LIN {X 0,Y 523.94,Z 179.22,A -85,B 0,C 180,E1 -4815.311,E2 -4815.311} C_VEL
LIN {X 0,Y 523.942,Z 179.221,A -85,B 0,C 180,E1 -4818.692,E2 -4818.692} C_VEL
LIN {X 0,Y 523.916,Z 179.219,A -85,B 0,C 180,E1 -4821.898,E2 -4821.898} C_VEL
LIN {X 0,Y 523.925,Z 179.226,A -85,B 0,C 180,E1 -4824.911,E2 -4824.911} C_VEL
LIN {X 0,Y 523.936,Z 179.217,A -85,B 0,C 180,E1 -4827.68,E2 -4827.68} C_VEL
LIN {X 0,Y 523.955,Z 179.221,A -85,B 0,C 180,E1 -4830.677,E2 -4830.677} C_VEL
LIN {X 0,Y 523.973,Z 179.213,A -85,B 0,C 180,E1 -4833.728,E2 -4833.728} C_VEL
LIN {X 0,Y 523.914,Z 179.223,A -85,B 0,C 180,E1 -4836.269,E2 -4836.269} C_VEL
LIN {X 0,Y 523.947,Z 179.222,A -85,B 0,C 180,E1 -4838.766,E2 -4838.766} C_VEL
LIN {X 0,Y 523.941,Z 179.218,A -85,B 0,C 180,E1 -4841.22,E2 -4841.22} C_VEL
LIN {X 0,Y 523.928,Z 179.219,A -85,B 0,C 180,E1 -4843.638,E2 -4843.638} C_VEL
LIN {X 0,Y 523.935,Z 179.221,A -85,B 0,C 180,E1 -4846.028,E2 -4846.028} C_VEL
LIN {X 0,Y 523.995,Z 179.211,A -85,B 0,C 180,E1 -4849.177,E2 -4849.177} C_VEL
LIN {X 0,Y 524.008,Z 179.216,A -85,B 0,C 180,E1 -4852.292,E2 -4852.292} C_VEL
LIN {X 0,Y 524.075,Z 179.206,A -85,B 0,C 180,E1 -4854.613,E2 -4854.613} C_VEL
LIN {X 0,Y 524.109,Z 179.2,A -85,B 0,C 180,E1 -4857.694,E2 -4857.694} C_VEL
LIN {X 0,Y 524.051,Z 179.302,A -85,B 0,C 180,E1 -4860.264,E2 -4860.264} C_VEL
LIN {X 0,Y 524.006,Z 197.303,A -85,B 0,C 180,E1 -4863.267,E2 -4863.267} C_VEL
LIN {X 0,Y 524.025,Z 211.019,A -85,B 0,C 180,E1 -4865.58,E2 -4865.58} C_VEL
LIN {X 0,Y 524.022,Z 224.908,A -85,B 0,C 180,E1 -4867.995,E2 -4867.995} C_VEL
LIN {X 0,Y 525.186,Z 232.663,A -85,B 0,C 180,E1 -4868.169,E2 -4868.169} C_VEL
LIN {X 0,Y 524.869,Z 303.638,A -85,B 0,C 180,E1 -4869.222,E2 -4869.222} C_VEL
LIN {X 0,Y 524.725,Z 315.282,A -85,B 0,C 180,E1 -4869.54,E2 -4869.54} C_VEL
LIN {X 0,Y 524.579,Z 326.858,A -85,B 0,C 180,E1 -4870.03,E2 -4870.03} C_VEL
LIN {X 0,Y 524.417,Z 337.03,A -85,B 0,C 180,E1 -4870.618,E2 -4870.618} C_VEL
LIN {X 0,Y 524.207,Z 347.39,A -85,B 0,C 180,E1 -4871.405,E2 -4871.405} C_VEL
LIN {X 0,Y 524.042,Z 355.429,A -85,B 0,C 180,E1 -4872.186,E2 -4872.186} C_VEL
LIN {X 0,Y 523.848,Z 363.637,A -85,B 0,C 180,E1 -4873.183,E2 -4873.183} C_VEL
LIN {X 0,Y 523.764,Z 370.012,A -85,B 0,C 180,E1 -4874.175,E2 -4874.175} C_VEL
LIN {X 0,Y 523.63,Z 375.152,A -85,B 0,C 180,E1 -4875.183,E2 -4875.183} C_VEL
LIN {X 0,Y 523.55,Z 379.695,A -85,B 0,C 180,E1 -4876.373,E2 -4876.373} C_VEL
LIN {X 0,Y 523.437,Z 382.89,A -85,B 0,C 180,E1 -4877.581,E2 -4877.581} C_VEL
LIN {X 0,Y 523.414,Z 384.762,A -85,B 0,C 180,E1 -4878.799,E2 -4878.799} C_VEL
LIN {X 0,Y 523.414,Z 385.391,A -85,B 0,C 180,E1 -4879.964,E2 -4879.964} C_VEL
LIN {X 0,Y 523.385,Z 384.744,A -85,B 0,C 180,E1 -4881.257,E2 -4881.257} C_VEL
LIN {X 0,Y 523.433,Z 383.554,A -85,B 0,C 180,E1 -4882.113,E2 -4882.113} C_VEL
LIN {X 0,Y 523.469,Z 380.727,A -85,B 0,C 180,E1 -4883.332,E2 -4883.332} C_VEL
LIN {X 0,Y 523.595,Z 376.321,A -85,B 0,C 180,E1 -4884.588,E2 -4884.588} C_VEL
LIN {X 0,Y 523.693,Z 371.04,A -85,B 0,C 180,E1 -4885.693,E2 -4885.693} C_VEL
LIN {X 0,Y 523.788,Z 364.719,A -85,B 0,C 180,E1 -4886.711,E2 -4886.711} C_VEL
LIN {X 0,Y 523.948,Z 356.846,A -85,B 0,C 180,E1 -4887.712,E2 -4887.712} C_VEL
LIN {X 0,Y 524.148,Z 347.477,A -85,B 0,C 180,E1 -4888.643,E2 -4888.643} C_VEL
LIN {X 0,Y 524.349,Z 337.621,A -85,B 0,C 180,E1 -4889.4,E2 -4889.4} C_VEL
LIN {X 0,Y 524.512,Z 327.606,A -85,B 0,C 180,E1 -4889.996,E2 -4889.996} C_VEL
LIN {X 0,Y 524.704,Z 315.795,A -85,B 0,C 180,E1 -4890.507,E2 -4890.507} C_VEL
LIN {X 0,Y 524.112,Z 310.181,A -85,B 0,C 180,E1 -4890.703,E2 -4890.703} C_VEL
LIN {X 0,Y 521.241,Z 300.997,A -85,B 0,C 180,E1 -4890.982,E2 -4890.982} C_VEL
LIN {X 0,Y 518.404,Z 291.68,A -85,B 0,C 180,E1 -4891.192,E2 -4891.192} C_VEL
LIN {X 0,Y 517.926,Z 285.863,A -85,B 0,C 180,E1 -4891.284,E2 -4891.284} C_VEL
LIN {X 0,Y 518.086,Z 231.937,A -85,B 0,C 180,E1 -4892.071,E2 -4892.071} C_VEL
LIN {X 0,Y 516.963,Z 225.027,A -85,B 0,C 180,E1 -4892.227,E2 -4892.227} C_VEL
LIN {X 0,Y 516.978,Z 220.993,A -85,B 0,C 180,E1 -4892.941,E2 -4892.941} C_VEL
LIN {X 0,Y 517.185,Z 204.967,A -85,B 0,C 180,E1 -4895.995,E2 -4895.995} C_VEL
LIN {X 0,Y 517.364,Z 187.914,A -85,B 0,C 180,E1 -4899.258,E2 -4899.258} C_VEL
LIN {X 0,Y 517.251,Z 181.728,A -85,B 0,C 180,E1 -4900.458,E2 -4900.458} C_VEL
LIN {X 0,Y 516.952,Z 180.119,A -85,B 0,C 180,E1 -4900.847,E2 -4900.847} C_VEL
LIN {X 0,Y 516.88,Z 180.104,A -85,B 0,C 180,E1 -4903.903,E2 -4903.903} C_VEL
LIN {X 0,Y 516.88,Z 180.101,A -85,B 0,C 180,E1 -4906.107,E2 -4906.107} C_VEL
LIN {X 0,Y 516.913,Z 180.092,A -85,B 0,C 180,E1 -4908.398,E2 -4908.398} C_VEL
LIN {X 0,Y 516.879,Z 180.099,A -85,B 0,C 180,E1 -4911.284,E2 -4911.284} C_VEL
LIN {X 0,Y 516.886,Z 180.096,A -85,B 0,C 180,E1 -4914.221,E2 -4914.221} C_VEL
LIN {X 0,Y 516.893,Z 180.095,A -85,B 0,C 180,E1 -4917.053,E2 -4917.053} C_VEL
LIN {X 0,Y 516.89,Z 180.099,A -85,B 0,C 180,E1 -4919.796,E2 -4919.796} C_VEL
LIN {X 0,Y 516.928,Z 180.089,A -85,B 0,C 180,E1 -4922.467,E2 -4922.467} C_VEL
LIN {X 0,Y 516.909,Z 180.095,A -85,B 0,C 180,E1 -4925.071,E2 -4925.071} C_VEL
LIN {X 0,Y 516.884,Z 180.094,A -85,B 0,C 180,E1 -4928.462,E2 -4928.462} C_VEL
LIN {X 0,Y 516.9,Z 180.096,A -85,B 0,C 180,E1 -4930.954,E2 -4930.954} C_VEL
LIN {X 0,Y 516.913,Z 180.099,A -85,B 0,C 180,E1 -4933.41,E2 -4933.41} C_VEL
LIN {X 0,Y 516.904,Z 180.094,A -85,B 0,C 180,E1 -4935.833,E2 -4935.833} C_VEL
LIN {X 0,Y 516.95,Z 180.092,A -85,B 0,C 180,E1 -4939.027,E2 -4939.027} C_VEL
LIN {X 0,Y 516.977,Z 180.083,A -85,B 0,C 180,E1 -4942.186,E2 -4942.186} C_VEL
LIN {X 0,Y 517.032,Z 180.077,A -85,B 0,C 180,E1 -4944.54,E2 -4944.54} C_VEL
LIN {X 0,Y 517.083,Z 180.072,A -85,B 0,C 180,E1 -4947.663,E2 -4947.663} C_VEL
LIN {X 0,Y 517.091,Z 180.073,A -85,B 0,C 180,E1 -4950.778,E2 -4950.778} C_VEL
LIN {X 0,Y 517.011,Z 180.087,A -85,B 0,C 180,E1 -4953.116,E2 -4953.116} C_VEL
LIN {X 0,Y 517,Z 180.081,A -85,B 0,C 180,E1 -4956.243,E2 -4956.243} C_VEL
LIN {X 0,Y 516.95,Z 180.089,A -85,B 0,C 180,E1 -4959.389,E2 -4959.389} C_VEL
LIN {X 0,Y 516.949,Z 180.086,A -85,B 0,C 180,E1 -4961.807,E2 -4961.807} C_VEL
LIN {X 0,Y 516.94,Z 180.092,A -85,B 0,C 180,E1 -4965.146,E2 -4965.146} C_VEL
LIN {X 0,Y 516.921,Z 180.092,A -85,B 0,C 180,E1 -4968.222,E2 -4968.222} C_VEL
LIN {X 0,Y 516.908,Z 180.1,A -85,B 0,C 180,E1 -4970.701,E2 -4970.701} C_VEL
LIN {X 0,Y 516.906,Z 180.093,A -85,B 0,C 180,E1 -4974.071,E2 -4974.071} C_VEL
LIN {X 0,Y 516.924,Z 180.099,A -85,B 0,C 180,E1 -4976.657,E2 -4976.657} C_VEL
LIN {X 0,Y 516.906,Z 180.092,A -85,B 0,C 180,E1 -4979.523,E2 -4979.523} C_VEL
LIN {X 0,Y 516.895,Z 180.102,A -85,B 0,C 180,E1 -4982.544,E2 -4982.544} C_VEL
LIN {X 0,Y 516.877,Z 180.096,A -85,B 0,C 180,E1 -4985.332,E2 -4985.332} C_VEL
LIN {X 0,Y 516.875,Z 180.098,A -85,B 0,C 180,E1 -4987.943,E2 -4987.943} C_VEL
LIN {X 0,Y 516.897,Z 180.098,A -85,B 0,C 180,E1 -4990.739,E2 -4990.739} C_VEL
LIN {X 0,Y 516.875,Z 180.098,A -85,B 0,C 180,E1 -4993.903,E2 -4993.903} C_VEL
LIN {X 0,Y 516.874,Z 180.101,A -85,B 0,C 180,E1 -4996.107,E2 -4996.107} C_VEL
LIN {X 0,Y 516.896,Z 180.093,A -85,B 0,C 180,E1 -4999.26,E2 -4999.26} C_VEL
LIN {X 0,Y 516.857,Z 180.107,A -85,B 0,C 180,E1 -5002.274,E2 -5002.274} C_VEL
LIN {X 0,Y 516.888,Z 180.094,A -85,B 0,C 180,E1 -5005.176,E2 -5005.176} C_VEL
LIN {X 0,Y 516.876,Z 180.102,A -85,B 0,C 180,E1 -5007.976,E2 -5007.976} C_VEL
LIN {X 0,Y 516.928,Z 180.091,A -85,B 0,C 180,E1 -5010.696,E2 -5010.696} C_VEL
LIN {X 0,Y 516.934,Z 180.093,A -85,B 0,C 180,E1 -5013.804,E2 -5013.804} C_VEL
LIN {X 0,Y 516.863,Z 180.098,A -85,B 0,C 180,E1 -5016.777,E2 -5016.777} C_VEL
LIN {X 0,Y 516.931,Z 180.094,A -85,B 0,C 180,E1 -5019.731,E2 -5019.731} C_VEL
LIN {X 0,Y 516.922,Z 180.091,A -85,B 0,C 180,E1 -5022.596,E2 -5022.596} C_VEL
LIN {X 0,Y 516.933,Z 180.089,A -85,B 0,C 180,E1 -5025.03,E2 -5025.03} C_VEL
LIN {X 0,Y 516.956,Z 180.089,A -85,B 0,C 180,E1 -5028.234,E2 -5028.234} C_VEL
LIN {X 0,Y 516.961,Z 180.088,A -85,B 0,C 180,E1 -5031.4,E2 -5031.4} C_VEL
LIN {X 0,Y 517,Z 180.089,A -85,B 0,C 180,E1 -5033.757,E2 -5033.757} C_VEL
LIN {X 0,Y 517.074,Z 180.079,A -85,B 0,C 180,E1 -5037.663,E2 -5037.663} C_VEL
LIN {X 0,Y 517.085,Z 180.069,A -85,B 0,C 180,E1 -5040.779,E2 -5040.779} C_VEL
LIN {X 0,Y 517.006,Z 180.082,A -85,B 0,C 180,E1 -5043.117,E2 -5043.117} C_VEL
LIN {X 0,Y 516.994,Z 180.082,A -85,B 0,C 180,E1 -5046.244,E2 -5046.244} C_VEL
LIN {X 0,Y 516.941,Z 180.094,A -85,B 0,C 180,E1 -5049.39,E2 -5049.39} C_VEL
LIN {X 0,Y 516.944,Z 180.091,A -85,B 0,C 180,E1 -5051.807,E2 -5051.807} C_VEL
LIN {X 0,Y 516.937,Z 180.093,A -85,B 0,C 180,E1 -5055.147,E2 -5055.147} C_VEL
LIN {X 0,Y 516.917,Z 180.091,A -85,B 0,C 180,E1 -5058.223,E2 -5058.223} C_VEL
LIN {X 0,Y 516.905,Z 180.093,A -85,B 0,C 180,E1 -5060.702,E2 -5060.702} C_VEL
LIN {X 0,Y 516.884,Z 180.095,A -85,B 0,C 180,E1 -5064.074,E2 -5064.074} C_VEL
LIN {X 0,Y 516.917,Z 180.092,A -85,B 0,C 180,E1 -5066.659,E2 -5066.659} C_VEL
LIN {X 0,Y 516.903,Z 180.097,A -85,B 0,C 180,E1 -5069.524,E2 -5069.524} C_VEL
LIN {X 0,Y 516.888,Z 180.095,A -85,B 0,C 180,E1 -5072.544,E2 -5072.544} C_VEL
LIN {X 0,Y 516.86,Z 180.103,A -85,B 0,C 180,E1 -5075.33,E2 -5075.33} C_VEL
LIN {X 0,Y 516.874,Z 180.096,A -85,B 0,C 180,E1 -5077.944,E2 -5077.944} C_VEL
LIN {X 0,Y 516.878,Z 180.1,A -85,B 0,C 180,E1 -5080.743,E2 -5080.743} C_VEL
LIN {X 0,Y 516.878,Z 180.102,A -85,B 0,C 180,E1 -5082.832,E2 -5082.832} C_VEL
LIN {X 0,Y 516.919,Z 180.099,A -85,B 0,C 180,E1 -5085.011,E2 -5085.011} C_VEL
LIN {X 0,Y 516.899,Z 180.095,A -85,B 0,C 180,E1 -5088.401,E2 -5088.401} C_VEL
LIN {X 0,Y 516.877,Z 180.099,A -85,B 0,C 180,E1 -5091.285,E2 -5091.285} C_VEL
LIN {X 0,Y 516.865,Z 180.098,A -85,B 0,C 180,E1 -5094.22,E2 -5094.22} C_VEL
LIN {X 0,Y 516.893,Z 180.101,A -85,B 0,C 180,E1 -5097.054,E2 -5097.054} C_VEL
LIN {X 0,Y 516.881,Z 180.098,A -85,B 0,C 180,E1 -5099.797,E2 -5099.797} C_VEL
LIN {X 0,Y 516.898,Z 180.101,A -85,B 0,C 180,E1 -5102.467,E2 -5102.467} C_VEL
LIN {X 0,Y 516.915,Z 180.238,A -85,B 0,C 180,E1 -5104.05,E2 -5104.05} C_VEL
LIN {X 0,Y 519.406,Z 191.693,A -85,B 0,C 180,E1 -5105.627,E2 -5105.627} C_VEL
LIN {X 0,Y 518.761,Z 215.518,A -85,B 0,C 180,E1 -5108.545,E2 -5108.545} C_VEL
LIN {X 0,Y 518.012,Z 242.728,A -85,B 0,C 180,E1 -5111.818,E2 -5111.818} C_VEL
LIN {X 0,Y 517.52,Z 267.094,A -85,B 0,C 180,E1 -5114.703,E2 -5114.703} C_VEL
LIN {X 0,Y 518.203,Z 273.127,A -85,B 0,C 180,E1 -5114.84,E2 -5114.84} C_VEL
LIN {X 0,Y 518.795,Z 280.471,A -85,B 0,C 180,E1 -5114.962,E2 -5114.962} C_VEL
LIN {X 0,Y 518.343,Z 376.522,A -85,B 0,C 180,E1 -5116.325,E2 -5116.325} C_VEL
LIN {X 0,Y 518.146,Z 389.838,A -85,B 0,C 180,E1 -5116.669,E2 -5116.669} C_VEL
LIN {X 0,Y 517.889,Z 402.606,A -85,B 0,C 180,E1 -5117.161,E2 -5117.161} C_VEL
LIN {X 0,Y 517.597,Z 414.328,A -85,B 0,C 180,E1 -5117.777,E2 -5117.777} C_VEL
LIN {X 0,Y 517.332,Z 425.652,A -85,B 0,C 180,E1 -5118.541,E2 -5118.541} C_VEL
LIN {X 0,Y 517.043,Z 436.193,A -85,B 0,C 180,E1 -5119.427,E2 -5119.427} C_VEL
LIN {X 0,Y 516.816,Z 445.668,A -85,B 0,C 180,E1 -5120.411,E2 -5120.411} C_VEL
LIN {X 0,Y 516.626,Z 454.821,A -85,B 0,C 180,E1 -5121.592,E2 -5121.592} C_VEL
LIN {X 0,Y 516.502,Z 462.192,A -85,B 0,C 180,E1 -5122.77,E2 -5122.77} C_VEL
LIN {X 0,Y 516.383,Z 467.166,A -85,B 0,C 180,E1 -5123.75,E2 -5123.75} C_VEL
LIN {X 0,Y 516.312,Z 471.994,A -85,B 0,C 180,E1 -5124.925,E2 -5124.925} C_VEL
LIN {X 0,Y 516.372,Z 475.691,A -85,B 0,C 180,E1 -5126.099,E2 -5126.099} C_VEL
LIN {X 0,Y 516.382,Z 477.594,A -85,B 0,C 180,E1 -5126.88,E2 -5126.88} C_VEL
LIN {X 0,Y 516.272,Z 479.011,A -85,B 0,C 180,E1 -5127.66,E2 -5127.66} C_VEL
LIN {X 0,Y 516.23,Z 480.634,A -85,B 0,C 180,E1 -5129.221,E2 -5129.221} C_VEL
LIN {X 0,Y 516.235,Z 480.847,A -85,B 0,C 180,E1 -5130.001,E2 -5130.001} C_VEL
LIN {X 0,Y 516.231,Z 480.617,A -85,B 0,C 180,E1 -5130.781,E2 -5130.781} C_VEL
LIN {X 0,Y 516.235,Z 479.989,A -85,B 0,C 180,E1 -5131.561,E2 -5131.561} C_VEL
LIN {X 0,Y 516.275,Z 478.962,A -85,B 0,C 180,E1 -5132.341,E2 -5132.341} C_VEL
LIN {X 0,Y 516.383,Z 477.526,A -85,B 0,C 180,E1 -5133.121,E2 -5133.121} C_VEL
LIN {X 0,Y 516.365,Z 474.5,A -85,B 0,C 180,E1 -5134.294,E2 -5134.294} C_VEL
LIN {X 0,Y 516.4,Z 470.409,A -85,B 0,C 180,E1 -5135.467,E2 -5135.467} C_VEL
LIN {X 0,Y 516.442,Z 465.064,A -85,B 0,C 180,E1 -5136.656,E2 -5136.656} C_VEL
LIN {X 0,Y 516.544,Z 458.49,A -85,B 0,C 180,E1 -5137.82,E2 -5137.82} C_VEL
LIN {X 0,Y 516.707,Z 450.22,A -85,B 0,C 180,E1 -5138.999,E2 -5138.999} C_VEL
LIN {X 0,Y 516.865,Z 441.765,A -85,B 0,C 180,E1 -5139.984,E2 -5139.984} C_VEL
LIN {X 0,Y 517.179,Z 431.397,A -85,B 0,C 180,E1 -5140.968,E2 -5140.968} C_VEL
LIN {X 0,Y 517.443,Z 419.886,A -85,B 0,C 180,E1 -5141.839,E2 -5141.839} C_VEL
LIN {X 0,Y 517.699,Z 408.046,A -85,B 0,C 180,E1 -5142.545,E2 -5142.545} C_VEL
LIN {X 0,Y 518.002,Z 396.026,A -85,B 0,C 180,E1 -5143.086,E2 -5143.086} C_VEL
LIN {X 0,Y 518.211,Z 383,A -85,B 0,C 180,E1 -5143.505,E2 -5143.505} C_VEL
LIN {X 0,Y 518.386,Z 370.827,A -85,B 0,C 180,E1 -5143.75,E2 -5143.75} C_VEL
LIN {X 0,Y 518.619,Z 277.097,A -85,B 0,C 180,E1 -5145.075,E2 -5145.075} C_VEL
LIN {X 0,Y 517.474,Z 266.884,A -85,B 0,C 180,E1 -5145.268,E2 -5145.268} C_VEL
LIN {X 0,Y 517.95,Z 241.231,A -85,B 0,C 180,E1 -5148.227,E2 -5148.227} C_VEL
LIN {X 0,Y 518.556,Z 211.729,A -85,B 0,C 180,E1 -5151.674,E2 -5151.674} C_VEL
LIN {X 0,Y 518.97,Z 190.784,A -85,B 0,C 180,E1 -5154.152,E2 -5154.152} C_VEL
LIN {X 0,Y 516.921,Z 180.235,A -85,B 0,C 180,E1 -5155.533,E2 -5155.533} C_VEL
LIN {X 0,Y 516.855,Z 180.103,A -85,B 0,C 180,E1 -5158.419,E2 -5158.419} C_VEL
LIN {X 0,Y 516.89,Z 180.103,A -85,B 0,C 180,E1 -5161.11,E2 -5161.11} C_VEL
LIN {X 0,Y 516.888,Z 180.097,A -85,B 0,C 180,E1 -5163.962,E2 -5163.962} C_VEL
LIN {X 0,Y 516.856,Z 180.104,A -85,B 0,C 180,E1 -5166.748,E2 -5166.748} C_VEL
LIN {X 0,Y 516.861,Z 180.101,A -85,B 0,C 180,E1 -5169.724,E2 -5169.724} C_VEL
LIN {X 0,Y 516.887,Z 180.097,A -85,B 0,C 180,E1 -5171.778,E2 -5171.778} C_VEL
LIN {X 0,Y 516.898,Z 180.102,A -85,B 0,C 180,E1 -5175.007,E2 -5175.007} C_VEL
LIN {X 0,Y 516.905,Z 180.094,A -85,B 0,C 180,E1 -5178.4,E2 -5178.4} C_VEL
LIN {X 0,Y 516.881,Z 180.099,A -85,B 0,C 180,E1 -5181.284,E2 -5181.284} C_VEL
LIN {X 0,Y 516.873,Z 180.098,A -85,B 0,C 180,E1 -5184.219,E2 -5184.219} C_VEL
LIN {X 0,Y 516.883,Z 180.101,A -85,B 0,C 180,E1 -5187.052,E2 -5187.052} C_VEL
LIN {X 0,Y 516.888,Z 180.095,A -85,B 0,C 180,E1 -5189.796,E2 -5189.796} C_VEL
LIN {X 0,Y 516.924,Z 180.097,A -85,B 0,C 180,E1 -5192.467,E2 -5192.467} C_VEL
LIN {X 0,Y 516.874,Z 180.1,A -85,B 0,C 180,E1 -5195.07,E2 -5195.07} C_VEL
LIN {X 0,Y 516.871,Z 180.097,A -85,B 0,C 180,E1 -5197.621,E2 -5197.621} C_VEL
LIN {X 0,Y 516.931,Z 180.093,A -85,B 0,C 180,E1 -5200.129,E2 -5200.129} C_VEL
LIN {X 0,Y 516.898,Z 180.101,A -85,B 0,C 180,E1 -5202.595,E2 -5202.595} C_VEL
LIN {X 0,Y 516.944,Z 180.091,A -85,B 0,C 180,E1 -5205.03,E2 -5205.03} C_VEL
LIN {X 0,Y 516.967,Z 180.091,A -85,B 0,C 180,E1 -5208.233,E2 -5208.233} C_VEL
LIN {X 0,Y 516.958,Z 180.087,A -85,B 0,C 180,E1 -5211.399,E2 -5211.399} C_VEL
LIN {X 0,Y 517.022,Z 180.085,A -85,B 0,C 180,E1 -5214.54,E2 -5214.54} C_VEL
LIN {X 0,Y 517.082,Z 180.075,A -85,B 0,C 180,E1 -5217.663,E2 -5217.663} C_VEL
LIN {X 0,Y 517.052,Z 180.202,A -85,B 0,C 180,E1 -5220.194,E2 -5220.194} C_VEL
LIN {X 0,Y 517.03,Z 199.023,A -85,B 0,C 180,E1 -5223.311,E2 -5223.311} C_VEL
LIN {X 0,Y 517.045,Z 214.996,A -85,B 0,C 180,E1 -5226.047,E2 -5226.047} C_VEL
LIN {X 0,Y 517.037,Z 224.992,A -85,B 0,C 180,E1 -5227.785,E2 -5227.785} C_VEL
LIN {X 0,Y 517.424,Z 227.519,A -85,B 0,C 180,E1 -5227.88,E2 -5227.88} C_VEL
LIN {X 0,Y 518.316,Z 234.268,A -85,B 0,C 180,E1 -5228.008,E2 -5228.008} C_VEL
LIN {X 0,Y 517.914,Z 304.483,A -85,B 0,C 180,E1 -5229.076,E2 -5229.076} C_VEL
LIN {X 0,Y 517.771,Z 316.676,A -85,B 0,C 180,E1 -5229.423,E2 -5229.423} C_VEL
LIN {X 0,Y 517.622,Z 328.964,A -85,B 0,C 180,E1 -5229.968,E2 -5229.968} C_VEL
LIN {X 0,Y 517.4,Z 340.176,A -85,B 0,C 180,E1 -5230.665,E2 -5230.665} C_VEL
LIN {X 0,Y 517.208,Z 349.918,A -85,B 0,C 180,E1 -5231.462,E2 -5231.462} C_VEL
LIN {X 0,Y 516.998,Z 358.584,A -85,B 0,C 180,E1 -5232.362,E2 -5232.362} C_VEL
LIN {X 0,Y 516.813,Z 366.175,A -85,B 0,C 180,E1 -5233.366,E2 -5233.366} C_VEL
LIN {X 0,Y 516.681,Z 372.203,A -85,B 0,C 180,E1 -5234.373,E2 -5234.373} C_VEL
LIN {X 0,Y 516.569,Z 376.772,A -85,B 0,C 180,E1 -5235.344,E2 -5235.344} C_VEL
LIN {X 0,Y 516.461,Z 381.227,A -85,B 0,C 180,E1 -5236.604,E2 -5236.604} C_VEL
LIN {X 0,Y 516.388,Z 383.835,A -85,B 0,C 180,E1 -5237.694,E2 -5237.694} C_VEL
LIN {X 0,Y 516.344,Z 385.689,A -85,B 0,C 180,E1 -5239.066,E2 -5239.066} C_VEL
LIN {X 0,Y 516.345,Z 386.049,A -85,B 0,C 180,E1 -5240.089,E2 -5240.089} C_VEL
LIN {X 0,Y 516.32,Z 385.831,A -85,B 0,C 180,E1 -5240.726,E2 -5240.726} C_VEL
LIN {X 0,Y 516.324,Z 385.075,A -85,B 0,C 180,E1 -5241.562,E2 -5241.562} C_VEL
LIN {X 0,Y 516.366,Z 383.7,A -85,B 0,C 180,E1 -5242.401,E2 -5242.401} C_VEL
LIN {X 0,Y 516.45,Z 380.478,A -85,B 0,C 180,E1 -5243.668,E2 -5243.668} C_VEL
LIN {X 0,Y 516.549,Z 375.681,A -85,B 0,C 180,E1 -5244.946,E2 -5244.946} C_VEL
LIN {X 0,Y 516.678,Z 369.555,A -85,B 0,C 180,E1 -5246.136,E2 -5246.136} C_VEL
LIN {X 0,Y 516.826,Z 363.178,A -85,B 0,C 180,E1 -5247.1,E2 -5247.1} C_VEL
LIN {X 0,Y 517.017,Z 354.953,A -85,B 0,C 180,E1 -5248.086,E2 -5248.086} C_VEL
LIN {X 0,Y 517.206,Z 345.75,A -85,B 0,C 180,E1 -5248.952,E2 -5248.952} C_VEL
LIN {X 0,Y 517.461,Z 335.624,A -85,B 0,C 180,E1 -5249.695,E2 -5249.695} C_VEL
LIN {X 0,Y 517.642,Z 324.246,A -85,B 0,C 180,E1 -5250.324,E2 -5250.324} C_VEL
LIN {X 0,Y 517.787,Z 312.012,A -85,B 0,C 180,E1 -5250.794,E2 -5250.794} C_VEL
LIN {X 0,Y 517.861,Z 300.164,A -85,B 0,C 180,E1 -5251.074,E2 -5251.074} C_VEL
LIN {X 0,Y 517.926,Z 285.863,A -85,B 0,C 180,E1 -5251.284,E2 -5251.284} C_VEL
LIN {X 0,Y 517.466,Z 280.046,A -85,B 0,C 180,E1 -5251.379,E2 -5251.379} C_VEL
LIN {X 0,Y 514.659,Z 270.702,A -85,B 0,C 180,E1 -5251.584,E2 -5251.584} C_VEL
LIN {X 0,Y 511.765,Z 261.363,A -85,B 0,C 180,E1 -5251.796,E2 -5251.796} C_VEL
LIN {X 0,Y 511.163,Z 255.544,A -85,B 0,C 180,E1 -5251.899,E2 -5251.899} C_VEL
LIN {X 0,Y 511.211,Z 232.848,A -85,B 0,C 180,E1 -5252.241,E2 -5252.241} C_VEL
LIN {X 0,Y 509.952,Z 225.174,A -85,B 0,C 180,E1 -5252.418,E2 -5252.418} C_VEL
LIN {X 0,Y 510.076,Z 210.803,A -85,B 0,C 180,E1 -5255.116,E2 -5255.116} C_VEL
LIN {X 0,Y 510.248,Z 196.891,A -85,B 0,C 180,E1 -5257.792,E2 -5257.792} C_VEL
LIN {X 0,Y 510.38,Z 183.783,A -85,B 0,C 180,E1 -5260.33,E2 -5260.33} C_VEL
LIN {X 0,Y 509.903,Z 181,A -85,B 0,C 180,E1 -5260.945,E2 -5260.945} C_VEL
LIN {X 0,Y 509.82,Z 180.98,A -85,B 0,C 180,E1 -5264.206,E2 -5264.206} C_VEL
LIN {X 0,Y 509.821,Z 180.976,A -85,B 0,C 180,E1 -5266.937,E2 -5266.937} C_VEL
LIN {X 0,Y 509.837,Z 180.98,A -85,B 0,C 180,E1 -5269.617,E2 -5269.617} C_VEL
LIN {X 0,Y 509.817,Z 180.975,A -85,B 0,C 180,E1 -5272.659,E2 -5272.659} C_VEL
LIN {X 0,Y 509.858,Z 180.976,A -85,B 0,C 180,E1 -5275.796,E2 -5275.796} C_VEL
LIN {X 0,Y 509.844,Z 180.972,A -85,B 0,C 180,E1 -5278.72,E2 -5278.72} C_VEL
LIN {X 0,Y 509.897,Z 180.968,A -85,B 0,C 180,E1 -5281.899,E2 -5281.899} C_VEL
LIN {X 0,Y 509.876,Z 180.968,A -85,B 0,C 180,E1 -5284.704,E2 -5284.704} C_VEL
LIN {X 0,Y 509.825,Z 180.983,A -85,B 0,C 180,E1 -5287.457,E2 -5287.457} C_VEL
LIN {X 0,Y 509.915,Z 180.965,A -85,B 0,C 180,E1 -5289.844,E2 -5289.844} C_VEL
LIN {X 0,Y 509.881,Z 180.973,A -85,B 0,C 180,E1 -5293.174,E2 -5293.174} C_VEL
LIN {X 0,Y 509.872,Z 180.972,A -85,B 0,C 180,E1 -5295.634,E2 -5295.634} C_VEL
LIN {X 0,Y 509.912,Z 180.967,A -85,B 0,C 180,E1 -5298.874,E2 -5298.874} C_VEL
LIN {X 0,Y 509.95,Z 180.958,A -85,B 0,C 180,E1 -5302.078,E2 -5302.078} C_VEL
LIN {X 0,Y 509.983,Z 180.955,A -85,B 0,C 180,E1 -5304.464,E2 -5304.464} C_VEL
LIN {X 0,Y 510.054,Z 180.947,A -85,B 0,C 180,E1 -5307.63,E2 -5307.63} C_VEL
LIN {X 0,Y 510.061,Z 180.949,A -85,B 0,C 180,E1 -5310.789,E2 -5310.789} C_VEL
LIN {X 0,Y 509.953,Z 180.965,A -85,B 0,C 180,E1 -5313.16,E2 -5313.16} C_VEL
LIN {X 0,Y 509.951,Z 180.959,A -85,B 0,C 180,E1 -5316.329,E2 -5316.329} C_VEL
LIN {X 0,Y 509.912,Z 180.969,A -85,B 0,C 180,E1 -5318.72,E2 -5318.72} C_VEL
LIN {X 0,Y 509.901,Z 180.964,A -85,B 0,C 180,E1 -5321.931,E2 -5321.931} C_VEL
LIN {X 0,Y 509.89,Z 180.969,A -85,B 0,C 180,E1 -5325.241,E2 -5325.241} C_VEL
LIN {X 0,Y 509.884,Z 180.967,A -85,B 0,C 180,E1 -5328,E2 -5328} C_VEL
LIN {X 0,Y 509.846,Z 180.977,A -85,B 0,C 180,E1 -5331.001,E2 -5331.001} C_VEL
LIN {X 0,Y 509.832,Z 180.973,A -85,B 0,C 180,E1 -5333.562,E2 -5333.562} C_VEL
LIN {X 0,Y 509.908,Z 180.968,A -85,B 0,C 180,E1 -5336.379,E2 -5336.379} C_VEL
LIN {X 0,Y 509.872,Z 180.974,A -85,B 0,C 180,E1 -5338.844,E2 -5338.844} C_VEL
LIN {X 0,Y 509.819,Z 180.975,A -85,B 0,C 180,E1 -5341.589,E2 -5341.589} C_VEL
LIN {X 0,Y 509.848,Z 180.978,A -85,B 0,C 180,E1 -5344.413,E2 -5344.413} C_VEL
LIN {X 0,Y 509.813,Z 180.976,A -85,B 0,C 180,E1 -5347.34,E2 -5347.34} C_VEL
LIN {X 0,Y 509.854,Z 180.978,A -85,B 0,C 180,E1 -5350.379,E2 -5350.379} C_VEL
LIN {X 0,Y 509.832,Z 180.974,A -85,B 0,C 180,E1 -5353.064,E2 -5353.064} C_VEL
LIN {X 0,Y 509.822,Z 180.976,A -85,B 0,C 180,E1 -5355.792,E2 -5355.792} C_VEL
LIN {X 0,Y 509.857,Z 180.975,A -85,B 0,C 180,E1 -5358.575,E2 -5358.575} C_VEL
LIN {X 0,Y 509.844,Z 180.974,A -85,B 0,C 180,E1 -5361.786,E2 -5361.786} C_VEL
LIN {X 0,Y 509.838,Z 180.976,A -85,B 0,C 180,E1 -5364.623,E2 -5364.623} C_VEL
LIN {X 0,Y 509.858,Z 180.971,A -85,B 0,C 180,E1 -5367.481,E2 -5367.481} C_VEL
LIN {X 0,Y 509.873,Z 180.975,A -85,B 0,C 180,E1 -5370.269,E2 -5370.269} C_VEL
LIN {X 0,Y 509.877,Z 180.968,A -85,B 0,C 180,E1 -5372.944,E2 -5372.944} C_VEL
LIN {X 0,Y 509.861,Z 180.972,A -85,B 0,C 180,E1 -5375.574,E2 -5375.574} C_VEL
LIN {X 0,Y 509.815,Z 180.982,A -85,B 0,C 180,E1 -5378.149,E2 -5378.149} C_VEL
LIN {X 0,Y 509.856,Z 180.971,A -85,B 0,C 180,E1 -5380.682,E2 -5380.682} C_VEL
LIN {X 0,Y 509.878,Z 180.968,A -85,B 0,C 180,E1 -5383.175,E2 -5383.175} C_VEL
LIN {X 0,Y 509.855,Z 180.975,A -85,B 0,C 180,E1 -5385.634,E2 -5385.634} C_VEL
LIN {X 0,Y 509.909,Z 180.963,A -85,B 0,C 180,E1 -5388.875,E2 -5388.875} C_VEL
LIN {X 0,Y 509.943,Z 180.964,A -85,B 0,C 180,E1 -5392.079,E2 -5392.079} C_VEL
LIN {X 0,Y 509.973,Z 180.956,A -85,B 0,C 180,E1 -5394.465,E2 -5394.465} C_VEL
LIN {X 0,Y 510.045,Z 180.954,A -85,B 0,C 180,E1 -5397.631,E2 -5397.631} C_VEL
LIN {X 0,Y 510.046,Z 180.951,A -85,B 0,C 180,E1 -5400,E2 -5400} C_VEL
LIN {X 0,Y 510.045,Z 180.947,A -85,B 0,C 180,E1 -5402.37,E2 -5402.37} C_VEL
LIN {X 0,Y 509.97,Z 180.964,A -85,B 0,C 180,E1 -5405.536,E2 -5405.536} C_VEL
LIN {X 0,Y 509.942,Z 180.963,A -85,B 0,C 180,E1 -5407.922,E2 -5407.922} C_VEL
LIN {X 0,Y 509.905,Z 180.968,A -85,B 0,C 180,E1 -5411.126,E2 -5411.126} C_VEL
LIN {X 0,Y 509.855,Z 180.97,A -85,B 0,C 180,E1 -5414.367,E2 -5414.367} C_VEL
LIN {X 0,Y 509.886,Z 180.972,A -85,B 0,C 180,E1 -5417.652,E2 -5417.652} C_VEL
LIN {X 0,Y 509.879,Z 180.967,A -85,B 0,C 180,E1 -5420.402,E2 -5420.402} C_VEL
LIN {X 0,Y 509.816,Z 180.98,A -85,B 0,C 180,E1 -5423.565,E2 -5423.565} C_VEL
LIN {X 0,Y 509.904,Z 180.964,A -85,B 0,C 180,E1 -5426.379,E2 -5426.379} C_VEL
LIN {X 0,Y 509.865,Z 180.972,A -85,B 0,C 180,E1 -5428.845,E2 -5428.845} C_VEL
LIN {X 0,Y 509.814,Z 180.979,A -85,B 0,C 180,E1 -5431.591,E2 -5431.591} C_VEL
LIN {X 0,Y 509.832,Z 180.974,A -85,B 0,C 180,E1 -5434.415,E2 -5434.415} C_VEL
LIN {X 0,Y 509.811,Z 180.981,A -85,B 0,C 180,E1 -5437.342,E2 -5437.342} C_VEL
LIN {X 0,Y 509.833,Z 180.974,A -85,B 0,C 180,E1 -5440.383,E2 -5440.383} C_VEL
LIN {X 0,Y 509.819,Z 180.983,A -85,B 0,C 180,E1 -5443.063,E2 -5443.063} C_VEL
LIN {X 0,Y 509.826,Z 180.974,A -85,B 0,C 180,E1 -5445.793,E2 -5445.793} C_VEL
LIN {X 0,Y 509.842,Z 180.976,A -85,B 0,C 180,E1 -5448.574,E2 -5448.574} C_VEL
LIN {X 0,Y 509.847,Z 180.971,A -85,B 0,C 180,E1 -5451.788,E2 -5451.788} C_VEL
LIN {X 0,Y 509.825,Z 180.98,A -85,B 0,C 180,E1 -5454.623,E2 -5454.623} C_VEL
LIN {X 0,Y 509.859,Z 180.973,A -85,B 0,C 180,E1 -5457.482,E2 -5457.482} C_VEL
LIN {X 0,Y 509.856,Z 180.976,A -85,B 0,C 180,E1 -5460.275,E2 -5460.275} C_VEL
LIN {X 0,Y 509.858,Z 180.977,A -85,B 0,C 180,E1 -5462.944,E2 -5462.944} C_VEL
LIN {X 0,Y 509.899,Z 181.21,A -85,B 0,C 180,E1 -5463.857,E2 -5463.857} C_VEL
LIN {X 0,Y 512.536,Z 193.358,A -85,B 0,C 180,E1 -5465.539,E2 -5465.539} C_VEL
LIN {X 0,Y 511.827,Z 216.977,A -85,B 0,C 180,E1 -5468.472,E2 -5468.472} C_VEL
LIN {X 0,Y 511.012,Z 245.942,A -85,B 0,C 180,E1 -5472.004,E2 -5472.004} C_VEL
LIN {X 0,Y 510.552,Z 267.228,A -85,B 0,C 180,E1 -5474.537,E2 -5474.537} C_VEL
LIN {X 0,Y 511.913,Z 279.701,A -85,B 0,C 180,E1 -5474.769,E2 -5474.769} C_VEL
LIN {X 0,Y 511.401,Z 376.087,A -85,B 0,C 180,E1 -5476.161,E2 -5476.161} C_VEL
LIN {X 0,Y 511.168,Z 389.375,A -85,B 0,C 180,E1 -5476.509,E2 -5476.509} C_VEL
LIN {X 0,Y 510.909,Z 401.56,A -85,B 0,C 180,E1 -5476.983,E2 -5476.983} C_VEL
LIN {X 0,Y 510.627,Z 412.709,A -85,B 0,C 180,E1 -5477.563,E2 -5477.563} C_VEL
LIN {X 0,Y 510.326,Z 424.822,A -85,B 0,C 180,E1 -5478.381,E2 -5478.381} C_VEL
LIN {X 0,Y 510.018,Z 435.409,A -85,B 0,C 180,E1 -5479.28,E2 -5479.28} C_VEL
LIN {X 0,Y 509.747,Z 444.931,A -85,B 0,C 180,E1 -5480.277,E2 -5480.277} C_VEL
LIN {X 0,Y 509.549,Z 454.109,A -85,B 0,C 180,E1 -5481.474,E2 -5481.474} C_VEL
LIN {X 0,Y 509.424,Z 461.501,A -85,B 0,C 180,E1 -5482.669,E2 -5482.669} C_VEL
LIN {X 0,Y 509.308,Z 466.492,A -85,B 0,C 180,E1 -5483.663,E2 -5483.663} C_VEL
LIN {X 0,Y 509.245,Z 471.333,A -85,B 0,C 180,E1 -5484.854,E2 -5484.854} C_VEL
LIN {X 0,Y 509.304,Z 475.039,A -85,B 0,C 180,E1 -5486.044,E2 -5486.044} C_VEL
LIN {X 0,Y 509.321,Z 476.946,A -85,B 0,C 180,E1 -5486.837,E2 -5486.837} C_VEL
LIN {X 0,Y 509.204,Z 478.367,A -85,B 0,C 180,E1 -5487.628,E2 -5487.628} C_VEL
LIN {X 0,Y 509.158,Z 479.988,A -85,B 0,C 180,E1 -5489.21,E2 -5489.21} C_VEL
LIN {X 0,Y 509.165,Z 480.2,A -85,B 0,C 180,E1 -5490.001,E2 -5490.001} C_VEL
LIN {X 0,Y 509.16,Z 479.967,A -85,B 0,C 180,E1 -5490.791,E2 -5490.791} C_VEL
LIN {X 0,Y 509.163,Z 479.333,A -85,B 0,C 180,E1 -5491.582,E2 -5491.582} C_VEL
LIN {X 0,Y 509.206,Z 478.3,A -85,B 0,C 180,E1 -5492.374,E2 -5492.374} C_VEL
LIN {X 0,Y 509.321,Z 476.857,A -85,B 0,C 180,E1 -5493.165,E2 -5493.165} C_VEL
LIN {X 0,Y 509.289,Z 473.816,A -85,B 0,C 180,E1 -5494.353,E2 -5494.353} C_VEL
LIN {X 0,Y 509.334,Z 469.707,A -85,B 0,C 180,E1 -5495.543,E2 -5495.543} C_VEL
LIN {X 0,Y 509.403,Z 463.483,A -85,B 0,C 180,E1 -5496.914,E2 -5496.914} C_VEL
LIN {X 0,Y 509.491,Z 456.469,A -85,B 0,C 180,E1 -5498.129,E2 -5498.129} C_VEL
LIN {X 0,Y 509.668,Z 447.88,A -85,B 0,C 180,E1 -5499.325,E2 -5499.325} C_VEL
LIN {X 0,Y 509.912,Z 438.023,A -85,B 0,C 180,E1 -5500.423,E2 -5500.423} C_VEL
LIN {X 0,Y 510.223,Z 428.109,A -85,B 0,C 180,E1 -5501.32,E2 -5501.32} C_VEL
LIN {X 0,Y 510.404,Z 416.923,A -85,B 0,C 180,E1 -5502.139,E2 -5502.139} C_VEL
LIN {X 0,Y 510.736,Z 404.941,A -85,B 0,C 180,E1 -5502.82,E2 -5502.82} C_VEL
LIN {X 0,Y 511.07,Z 392.118,A -85,B 0,C 180,E1 -5503.368,E2 -5503.368} C_VEL
LIN {X 0,Y 511.338,Z 379.376,A -85,B 0,C 180,E1 -5503.741,E2 -5503.741} C_VEL
LIN {X 0,Y 511.482,Z 361.33,A -85,B 0,C 180,E1 -5504.041,E2 -5504.041} C_VEL
LIN {X 0,Y 511.758,Z 277.955,A -85,B 0,C 180,E1 -5505.24,E2 -5505.24} C_VEL
LIN {X 0,Y 510.448,Z 266.463,A -85,B 0,C 180,E1 -5505.467,E2 -5505.467} C_VEL
LIN {X 0,Y 510.959,Z 241.001,A -85,B 0,C 180,E1 -5508.443,E2 -5508.443} C_VEL
LIN {X 0,Y 511.619,Z 212.915,A -85,B 0,C 180,E1 -5511.771,E2 -5511.771} C_VEL
LIN {X 0,Y 512.045,Z 191.704,A -85,B 0,C 180,E1 -5514.316,E2 -5514.316} C_VEL
LIN {X 0,Y 509.872,Z 181.114,A -85,B 0,C 180,E1 -5515.734,E2 -5515.734} C_VEL
LIN {X 0,Y 509.841,Z 180.979,A -85,B 0,C 180,E1 -5518.847,E2 -5518.847} C_VEL
LIN {X 0,Y 509.821,Z 180.981,A -85,B 0,C 180,E1 -5521.59,E2 -5521.59} C_VEL
LIN {X 0,Y 509.84,Z 180.976,A -85,B 0,C 180,E1 -5524.415,E2 -5524.415} C_VEL
LIN {X 0,Y 509.81,Z 180.983,A -85,B 0,C 180,E1 -5527.342,E2 -5527.342} C_VEL
LIN {X 0,Y 509.817,Z 180.978,A -85,B 0,C 180,E1 -5530.384,E2 -5530.384} C_VEL
LIN {X 0,Y 509.802,Z 180.985,A -85,B 0,C 180,E1 -5533.059,E2 -5533.059} C_VEL
LIN {X 0,Y 509.824,Z 180.975,A -85,B 0,C 180,E1 -5535.793,E2 -5535.793} C_VEL
LIN {X 0,Y 509.848,Z 180.975,A -85,B 0,C 180,E1 -5538.573,E2 -5538.573} C_VEL
LIN {X 0,Y 509.852,Z 180.971,A -85,B 0,C 180,E1 -5541.786,E2 -5541.786} C_VEL
LIN {X 0,Y 509.831,Z 180.979,A -85,B 0,C 180,E1 -5544.622,E2 -5544.622} C_VEL
LIN {X 0,Y 509.862,Z 180.971,A -85,B 0,C 180,E1 -5547.48,E2 -5547.48} C_VEL
LIN {X 0,Y 509.86,Z 180.974,A -85,B 0,C 180,E1 -5550.274,E2 -5550.274} C_VEL
LIN {X 0,Y 509.883,Z 180.973,A -85,B 0,C 180,E1 -5552.944,E2 -5552.944} C_VEL
LIN {X 0,Y 509.851,Z 180.972,A -85,B 0,C 180,E1 -5555.573,E2 -5555.573} C_VEL
LIN {X 0,Y 509.823,Z 180.978,A -85,B 0,C 180,E1 -5558.148,E2 -5558.148} C_VEL
LIN {X 0,Y 509.859,Z 180.977,A -85,B 0,C 180,E1 -5560.681,E2 -5560.681} C_VEL
LIN {X 0,Y 509.869,Z 180.971,A -85,B 0,C 180,E1 -5563.174,E2 -5563.174} C_VEL
LIN {X 0,Y 509.862,Z 180.971,A -85,B 0,C 180,E1 -5565.634,E2 -5565.634} C_VEL
LIN {X 0,Y 509.913,Z 180.968,A -85,B 0,C 180,E1 -5568.874,E2 -5568.874} C_VEL
LIN {X 0,Y 509.922,Z 180.969,A -85,B 0,C 180,E1 -5572.078,E2 -5572.078} C_VEL
LIN {X 0,Y 509.973,Z 180.964,A -85,B 0,C 180,E1 -5574.464,E2 -5574.464} C_VEL
LIN {X 0,Y 510.053,Z 180.951,A -85,B 0,C 180,E1 -5577.631,E2 -5577.631} C_VEL
LIN {X 0,Y 510.047,Z 181.174,A -85,B 0,C 180,E1 -5580.123,E2 -5580.123} C_VEL
LIN {X 0,Y 510.04,Z 199.4,A -85,B 0,C 180,E1 -5583.159,E2 -5583.159} C_VEL
LIN {X 0,Y 510.038,Z 215.703,A -85,B 0,C 180,E1 -5585.931,E2 -5585.931} C_VEL
LIN {X 0,Y 510.066,Z 225.334,A -85,B 0,C 180,E1 -5587.596,E2 -5587.596} C_VEL
LIN {X 0,Y 510.941,Z 230.568,A -85,B 0,C 180,E1 -5587.742,E2 -5587.742} C_VEL
LIN {X 0,Y 511.433,Z 234.837,A -85,B 0,C 180,E1 -5587.823,E2 -5587.823} C_VEL
LIN {X 0,Y 510.939,Z 305.417,A -85,B 0,C 180,E1 -5588.927,E2 -5588.927} C_VEL
LIN {X 0,Y 510.847,Z 316.696,A -85,B 0,C 180,E1 -5589.252,E2 -5589.252} C_VEL
LIN {X 0,Y 510.694,Z 327.176,A -85,B 0,C 180,E1 -5589.705,E2 -5589.705} C_VEL
LIN {X 0,Y 510.509,Z 337.57,A -85,B 0,C 180,E1 -5590.309,E2 -5590.309} C_VEL
LIN {X 0,Y 510.259,Z 348.071,A -85,B 0,C 180,E1 -5591.117,E2 -5591.117} C_VEL
LIN {X 0,Y 510.075,Z 356.683,A -85,B 0,C 180,E1 -5591.968,E2 -5591.968} C_VEL
LIN {X 0,Y 509.848,Z 364.56,A -85,B 0,C 180,E1 -5592.944,E2 -5592.944} C_VEL
LIN {X 0,Y 509.721,Z 371.025,A -85,B 0,C 180,E1 -5593.962,E2 -5593.962} C_VEL
LIN {X 0,Y 509.538,Z 377.076,A -85,B 0,C 180,E1 -5595.192,E2 -5595.192} C_VEL
LIN {X 0,Y 509.437,Z 381.49,A -85,B 0,C 180,E1 -5596.428,E2 -5596.428} C_VEL
LIN {X 0,Y 509.316,Z 384.744,A -85,B 0,C 180,E1 -5597.801,E2 -5597.801} C_VEL
LIN {X 0,Y 509.279,Z 385.809,A -85,B 0,C 180,E1 -5598.505,E2 -5598.505} C_VEL
LIN {X 0,Y 509.268,Z 386.513,A -85,B 0,C 180,E1 -5599.341,E2 -5599.341} C_VEL
LIN {X 0,Y 509.268,Z 386.673,A -85,B 0,C 180,E1 -5600.213,E2 -5600.213} C_VEL
LIN {X 0,Y 509.274,Z 386.287,A -85,B 0,C 180,E1 -5601.026,E2 -5601.026} C_VEL
LIN {X 0,Y 509.305,Z 384.396,A -85,B 0,C 180,E1 -5602.4,E2 -5602.4} C_VEL
LIN {X 0,Y 509.379,Z 381.516,A -85,B 0,C 180,E1 -5603.585,E2 -5603.585} C_VEL
LIN {X 0,Y 509.491,Z 376.855,A -85,B 0,C 180,E1 -5604.88,E2 -5604.88} C_VEL
LIN {X 0,Y 509.641,Z 371.576,A -85,B 0,C 180,E1 -5605.965,E2 -5605.965} C_VEL
LIN {X 0,Y 509.784,Z 364.728,A -85,B 0,C 180,E1 -5607.061,E2 -5607.061} C_VEL
LIN {X 0,Y 509.954,Z 357.808,A -85,B 0,C 180,E1 -5607.941,E2 -5607.941} C_VEL
LIN {X 0,Y 510.169,Z 349.137,A -85,B 0,C 180,E1 -5608.826,E2 -5608.826} C_VEL
LIN {X 0,Y 510.404,Z 339.47,A -85,B 0,C 180,E1 -5609.602,E2 -5609.602} C_VEL
LIN {X 0,Y 510.598,Z 328.832,A -85,B 0,C 180,E1 -5610.261,E2 -5610.261} C_VEL
LIN {X 0,Y 510.793,Z 317.413,A -85,B 0,C 180,E1 -5610.774,E2 -5610.774} C_VEL
LIN {X 0,Y 510.892,Z 306.341,A -85,B 0,C 180,E1 -5611.112,E2 -5611.112} C_VEL
LIN {X 0,Y 510.95,Z 287.551,A -85,B 0,C 180,E1 -5611.425,E2 -5611.425} C_VEL
LIN {X 0,Y 511.163,Z 255.544,A -85,B 0,C 180,E1 -5611.899,E2 -5611.899} C_VEL
LIN {X 0,Y 510.559,Z 251.663,A -85,B 0,C 180,E1 -5611.973,E2 -5611.973} C_VEL
LIN {X 0,Y 505.041,Z 239.67,A -85,B 0,C 180,E1 -5612.302,E2 -5612.302} C_VEL
LIN {X 0,Y 504.429,Z 235.789,A -85,B 0,C 180,E1 -5612.379,E2 -5612.379} C_VEL
LIN {X 0,Y 503.236,Z 227.287,A -85,B 0,C 180,E1 -5612.543,E2 -5612.543} C_VEL
LIN {X 0,Y 502.93,Z 225.116,A -85,B 0,C 180,E1 -5612.636,E2 -5612.636} C_VEL
LIN {X 0,Y 503.16,Z 208.044,A -85,B 0,C 180,E1 -5615.891,E2 -5615.891} C_VEL
LIN {X 0,Y 503.367,Z 192.403,A -85,B 0,C 180,E1 -5618.923,E2 -5618.923} C_VEL
LIN {X 0,Y 503.331,Z 184.57,A -85,B 0,C 180,E1 -5620.458,E2 -5620.458} C_VEL
LIN {X 0,Y 502.86,Z 181.871,A -85,B 0,C 180,E1 -5621.078,E2 -5621.078} C_VEL
LIN {X 0,Y 502.784,Z 181.854,A -85,B 0,C 180,E1 -5624.53,E2 -5624.53} C_VEL
LIN {X 0,Y 502.795,Z 181.858,A -85,B 0,C 180,E1 -5627.86,E2 -5627.86} C_VEL
LIN {X 0,Y 502.799,Z 181.85,A -85,B 0,C 180,E1 -5631.024,E2 -5631.024} C_VEL
LIN {X 0,Y 502.781,Z 181.853,A -85,B 0,C 180,E1 -5634.167,E2 -5634.167} C_VEL
LIN {X 0,Y 502.831,Z 181.847,A -85,B 0,C 180,E1 -5636.993,E2 -5636.993} C_VEL
LIN {X 0,Y 502.813,Z 181.849,A -85,B 0,C 180,E1 -5640.065,E2 -5640.065} C_VEL
LIN {X 0,Y 502.833,Z 181.845,A -85,B 0,C 180,E1 -5642.533,E2 -5642.533} C_VEL
LIN {X 0,Y 502.826,Z 181.852,A -85,B 0,C 180,E1 -5645.299,E2 -5645.299} C_VEL
LIN {X 0,Y 502.778,Z 181.855,A -85,B 0,C 180,E1 -5647.826,E2 -5647.826} C_VEL
LIN {X 0,Y 502.822,Z 181.846,A -85,B 0,C 180,E1 -5650.4,E2 -5650.4} C_VEL
LIN {X 0,Y 502.829,Z 181.849,A -85,B 0,C 180,E1 -5652.931,E2 -5652.931} C_VEL
LIN {X 0,Y 502.85,Z 181.85,A -85,B 0,C 180,E1 -5655.429,E2 -5655.429} C_VEL
LIN {X 0,Y 502.876,Z 181.841,A -85,B 0,C 180,E1 -5658.716,E2 -5658.716} C_VEL
LIN {X 0,Y 502.9,Z 181.837,A -85,B 0,C 180,E1 -5661.966,E2 -5661.966} C_VEL
LIN {X 0,Y 502.939,Z 181.832,A -85,B 0,C 180,E1 -5664.386,E2 -5664.386} C_VEL
LIN {X 0,Y 503.024,Z 181.824,A -85,B 0,C 180,E1 -5667.597,E2 -5667.597} C_VEL
LIN {X 0,Y 503.025,Z 181.821,A -85,B 0,C 180,E1 -5669.999,E2 -5669.999} C_VEL
LIN {X 0,Y 503.023,Z 181.822,A -85,B 0,C 180,E1 -5672.402,E2 -5672.402} C_VEL
LIN {X 0,Y 502.931,Z 181.834,A -85,B 0,C 180,E1 -5675.613,E2 -5675.613} C_VEL
LIN {X 0,Y 502.898,Z 181.837,A -85,B 0,C 180,E1 -5678.033,E2 -5678.033} C_VEL
LIN {X 0,Y 502.874,Z 181.843,A -85,B 0,C 180,E1 -5681.283,E2 -5681.283} C_VEL
LIN {X 0,Y 502.841,Z 181.849,A -85,B 0,C 180,E1 -5684.57,E2 -5684.57} C_VEL
LIN {X 0,Y 502.858,Z 181.842,A -85,B 0,C 180,E1 -5687.906,E2 -5687.906} C_VEL
LIN {X 0,Y 502.824,Z 181.852,A -85,B 0,C 180,E1 -5690.536,E2 -5690.536} C_VEL
LIN {X 0,Y 502.792,Z 181.854,A -85,B 0,C 180,E1 -5693.04,E2 -5693.04} C_VEL
LIN {X 0,Y 502.837,Z 181.844,A -85,B 0,C 180,E1 -5695.675,E2 -5695.675} C_VEL
LIN {X 0,Y 502.835,Z 181.85,A -85,B 0,C 180,E1 -5698.372,E2 -5698.372} C_VEL
LIN {X 0,Y 502.79,Z 181.85,A -85,B 0,C 180,E1 -5701.499,E2 -5701.499} C_VEL
LIN {X 0,Y 502.801,Z 181.856,A -85,B 0,C 180,E1 -5704.444,E2 -5704.444} C_VEL
LIN {X 0,Y 502.775,Z 181.853,A -85,B 0,C 180,E1 -5707.178,E2 -5707.178} C_VEL
LIN {X 0,Y 502.814,Z 181.85,A -85,B 0,C 180,E1 -5710.011,E2 -5710.011} C_VEL
LIN {X 0,Y 502.815,Z 181.853,A -85,B 0,C 180,E1 -5712.201,E2 -5712.201} C_VEL
LIN {X 0,Y 502.792,Z 181.85,A -85,B 0,C 180,E1 -5715.468,E2 -5715.468} C_VEL
LIN {X 0,Y 502.818,Z 181.848,A -85,B 0,C 180,E1 -5719.004,E2 -5719.004} C_VEL
LIN {X 0,Y 502.786,Z 181.856,A -85,B 0,C 180,E1 -5722.046,E2 -5722.046} C_VEL
LIN {X 0,Y 502.802,Z 181.849,A -85,B 0,C 180,E1 -5725.035,E2 -5725.035} C_VEL
LIN {X 0,Y 502.78,Z 181.856,A -85,B 0,C 180,E1 -5727.916,E2 -5727.916} C_VEL
LIN {X 0,Y 502.831,Z 181.847,A -85,B 0,C 180,E1 -5730.713,E2 -5730.713} C_VEL
LIN {X 0,Y 502.853,Z 181.843,A -85,B 0,C 180,E1 -5733.439,E2 -5733.439} C_VEL
LIN {X 0,Y 502.783,Z 181.86,A -85,B 0,C 180,E1 -5736.086,E2 -5736.086} C_VEL
LIN {X 0,Y 502.775,Z 181.853,A -85,B 0,C 180,E1 -5738.689,E2 -5738.689} C_VEL
LIN {X 0,Y 502.822,Z 181.847,A -85,B 0,C 180,E1 -5741.248,E2 -5741.248} C_VEL
LIN {X 0,Y 502.815,Z 181.854,A -85,B 0,C 180,E1 -5743.767,E2 -5743.767} C_VEL
LIN {X 0,Y 502.822,Z 181.85,A -85,B 0,C 180,E1 -5746.255,E2 -5746.255} C_VEL
LIN {X 0,Y 502.873,Z 181.84,A -85,B 0,C 180,E1 -5748.717,E2 -5748.717} C_VEL
LIN {X 0,Y 502.893,Z 181.844,A -85,B 0,C 180,E1 -5751.967,E2 -5751.967} C_VEL
LIN {X 0,Y 502.929,Z 181.834,A -85,B 0,C 180,E1 -5754.387,E2 -5754.387} C_VEL
LIN {X 0,Y 503.015,Z 181.829,A -85,B 0,C 180,E1 -5757.598,E2 -5757.598} C_VEL
LIN {X 0,Y 503.017,Z 181.826,A -85,B 0,C 180,E1 -5760,E2 -5760} C_VEL
LIN {X 0,Y 503.015,Z 181.823,A -85,B 0,C 180,E1 -5762.403,E2 -5762.403} C_VEL
LIN {X 0,Y 502.924,Z 181.842,A -85,B 0,C 180,E1 -5765.614,E2 -5765.614} C_VEL
LIN {X 0,Y 502.892,Z 181.84,A -85,B 0,C 180,E1 -5768.034,E2 -5768.034} C_VEL
LIN {X 0,Y 502.869,Z 181.846,A -85,B 0,C 180,E1 -5771.284,E2 -5771.284} C_VEL
LIN {X 0,Y 502.836,Z 181.845,A -85,B 0,C 180,E1 -5774.571,E2 -5774.571} C_VEL
LIN {X 0,Y 502.847,Z 181.845,A -85,B 0,C 180,E1 -5777.908,E2 -5777.908} C_VEL
LIN {X 0,Y 502.822,Z 181.847,A -85,B 0,C 180,E1 -5780.537,E2 -5780.537} C_VEL
LIN {X 0,Y 502.781,Z 181.856,A -85,B 0,C 180,E1 -5783.041,E2 -5783.041} C_VEL
LIN {X 0,Y 502.831,Z 181.848,A -85,B 0,C 180,E1 -5785.676,E2 -5785.676} C_VEL
LIN {X 0,Y 502.831,Z 181.845,A -85,B 0,C 180,E1 -5788.374,E2 -5788.374} C_VEL
LIN {X 0,Y 502.787,Z 181.855,A -85,B 0,C 180,E1 -5791.5,E2 -5791.5} C_VEL
LIN {X 0,Y 502.783,Z 181.851,A -85,B 0,C 180,E1 -5793.996,E2 -5793.996} C_VEL
LIN {X 0,Y 502.772,Z 181.86,A -85,B 0,C 180,E1 -5797.179,E2 -5797.179} C_VEL
LIN {X 0,Y 502.783,Z 181.851,A -85,B 0,C 180,E1 -5800.016,E2 -5800.016} C_VEL
LIN {X 0,Y 502.799,Z 181.849,A -85,B 0,C 180,E1 -5802.2,E2 -5802.2} C_VEL
LIN {X 0,Y 502.797,Z 181.852,A -85,B 0,C 180,E1 -5805.469,E2 -5805.469} C_VEL
LIN {X 0,Y 502.791,Z 181.85,A -85,B 0,C 180,E1 -5807.861,E2 -5807.861} C_VEL
LIN {X 0,Y 502.798,Z 181.856,A -85,B 0,C 180,E1 -5811.025,E2 -5811.025} C_VEL
LIN {X 0,Y 502.768,Z 181.854,A -85,B 0,C 180,E1 -5814.171,E2 -5814.171} C_VEL
LIN {X 0,Y 502.831,Z 181.853,A -85,B 0,C 180,E1 -5816.994,E2 -5816.994} C_VEL
LIN {X 0,Y 502.812,Z 181.852,A -85,B 0,C 180,E1 -5820.066,E2 -5820.066} C_VEL
LIN {X 0,Y 502.844,Z 181.899,A -85,B 0,C 180,E1 -5823.531,E2 -5823.531} C_VEL
LIN {X 0,Y 502.913,Z 182.245,A -85,B 0,C 180,E1 -5823.661,E2 -5823.661} C_VEL
LIN {X 0,Y 505.571,Z 194.276,A -85,B 0,C 180,E1 -5825.353,E2 -5825.353} C_VEL
LIN {X 0,Y 505.298,Z 206.579,A -85,B 0,C 180,E1 -5826.913,E2 -5826.913} C_VEL
LIN {X 0,Y 504.476,Z 229.98,A -85,B 0,C 180,E1 -5829.831,E2 -5829.831} C_VEL
LIN {X 0,Y 503.798,Z 255.433,A -85,B 0,C 180,E1 -5832.966,E2 -5832.966} C_VEL
LIN {X 0,Y 503.537,Z 266.783,A -85,B 0,C 180,E1 -5834.331,E2 -5834.331} C_VEL
LIN {X 0,Y 505,Z 280.63,A -85,B 0,C 180,E1 -5834.596,E2 -5834.596} C_VEL
LIN {X 0,Y 504.447,Z 375.649,A -85,B 0,C 180,E1 -5835.992,E2 -5835.992} C_VEL
LIN {X 0,Y 504.226,Z 388.918,A -85,B 0,C 180,E1 -5836.346,E2 -5836.346} C_VEL
LIN {X 0,Y 503.919,Z 401.653,A -85,B 0,C 180,E1 -5836.85,E2 -5836.85} C_VEL
LIN {X 0,Y 503.581,Z 413.483,A -85,B 0,C 180,E1 -5837.491,E2 -5837.491} C_VEL
LIN {X 0,Y 503.278,Z 425.297,A -85,B 0,C 180,E1 -5838.318,E2 -5838.318} C_VEL
LIN {X 0,Y 502.952,Z 435.698,A -85,B 0,C 180,E1 -5839.229,E2 -5839.229} C_VEL
LIN {X 0,Y 502.628,Z 445.845,A -85,B 0,C 180,E1 -5840.341,E2 -5840.341} C_VEL
LIN {X 0,Y 502.453,Z 454.774,A -85,B 0,C 180,E1 -5841.555,E2 -5841.555} C_VEL
LIN {X 0,Y 502.335,Z 461.895,A -85,B 0,C 180,E1 -5842.767,E2 -5842.767} C_VEL
LIN {X 0,Y 502.226,Z 467.576,A -85,B 0,C 180,E1 -5843.976,E2 -5843.976} C_VEL
LIN {X 0,Y 502.122,Z 472.026,A -85,B 0,C 180,E1 -5845.183,E2 -5845.183} C_VEL
LIN {X 0,Y 502.236,Z 474.386,A -85,B 0,C 180,E1 -5845.989,E2 -5845.989} C_VEL
LIN {X 0,Y 502.262,Z 476.298,A -85,B 0,C 180,E1 -5846.792,E2 -5846.792} C_VEL
LIN {X 0,Y 502.138,Z 477.722,A -85,B 0,C 180,E1 -5847.594,E2 -5847.594} C_VEL
LIN {X 0,Y 502.086,Z 479.342,A -85,B 0,C 180,E1 -5849.199,E2 -5849.199} C_VEL
LIN {X 0,Y 502.095,Z 479.553,A -85,B 0,C 180,E1 -5850.001,E2 -5850.001} C_VEL
LIN {X 0,Y 502.088,Z 479.317,A -85,B 0,C 180,E1 -5850.803,E2 -5850.803} C_VEL
LIN {X 0,Y 502.14,Z 477.639,A -85,B 0,C 180,E1 -5852.407,E2 -5852.407} C_VEL
LIN {X 0,Y 502.262,Z 476.188,A -85,B 0,C 180,E1 -5853.209,E2 -5853.209} C_VEL
LIN {X 0,Y 502.197,Z 473.13,A -85,B 0,C 180,E1 -5854.415,E2 -5854.415} C_VEL
LIN {X 0,Y 502.267,Z 469.005,A -85,B 0,C 180,E1 -5855.622,E2 -5855.622} C_VEL
LIN {X 0,Y 502.331,Z 462.75,A -85,B 0,C 180,E1 -5857.012,E2 -5857.012} C_VEL
LIN {X 0,Y 502.427,Z 455.709,A -85,B 0,C 180,E1 -5858.244,E2 -5858.244} C_VEL
LIN {X 0,Y 502.577,Z 447.071,A -85,B 0,C 180,E1 -5859.458,E2 -5859.458} C_VEL
LIN {X 0,Y 502.843,Z 438.171,A -85,B 0,C 180,E1 -5860.469,E2 -5860.469} C_VEL
LIN {X 0,Y 503.138,Z 427.201,A -85,B 0,C 180,E1 -5861.482,E2 -5861.482} C_VEL
LIN {X 0,Y 503.386,Z 416.523,A -85,B 0,C 180,E1 -5862.273,E2 -5862.273} C_VEL
LIN {X 0,Y 503.743,Z 404.849,A -85,B 0,C 180,E1 -5862.95,E2 -5862.95} C_VEL
LIN {X 0,Y 504.078,Z 392.18,A -85,B 0,C 180,E1 -5863.506,E2 -5863.506} C_VEL
LIN {X 0,Y 504.368,Z 379.903,A -85,B 0,C 180,E1 -5863.883,E2 -5863.883} C_VEL
LIN {X 0,Y 504.535,Z 364.299,A -85,B 0,C 180,E1 -5864.161,E2 -5864.161} C_VEL
LIN {X 0,Y 504.86,Z 278.555,A -85,B 0,C 180,E1 -5865.419,E2 -5865.419} C_VEL
LIN {X 0,Y 503.464,Z 266.006,A -85,B 0,C 180,E1 -5865.676,E2 -5865.676} C_VEL
LIN {X 0,Y 504.004,Z 240.42,A -85,B 0,C 180,E1 -5868.707,E2 -5868.707} C_VEL
LIN {X 0,Y 504.681,Z 214.131,A -85,B 0,C 180,E1 -5871.871,E2 -5871.871} C_VEL
LIN {X 0,Y 505.162,Z 194.661,A -85,B 0,C 180,E1 -5874.231,E2 -5874.231} C_VEL
LIN {X 0,Y 504.505,Z 189.674,A -85,B 0,C 180,E1 -5874.876,E2 -5874.876} C_VEL
LIN {X 0,Y 502.831,Z 181.97,A -85,B 0,C 180,E1 -5875.954,E2 -5875.954} C_VEL
LIN {X 0,Y 502.808,Z 181.857,A -85,B 0,C 180,E1 -5879.289,E2 -5879.289} C_VEL
LIN {X 0,Y 502.785,Z 181.854,A -85,B 0,C 180,E1 -5882.085,E2 -5882.085} C_VEL
LIN {X 0,Y 502.797,Z 181.857,A -85,B 0,C 180,E1 -5884.966,E2 -5884.966} C_VEL
LIN {X 0,Y 502.794,Z 181.853,A -85,B 0,C 180,E1 -5888.485,E2 -5888.485} C_VEL
LIN {X 0,Y 502.774,Z 181.86,A -85,B 0,C 180,E1 -5891.071,E2 -5891.071} C_VEL
LIN {X 0,Y 502.759,Z 181.859,A -85,B 0,C 180,E1 -5893.372,E2 -5893.372} C_VEL
LIN {X 0,Y 502.781,Z 181.853,A -85,B 0,C 180,E1 -5895.66,E2 -5895.66} C_VEL
LIN {X 0,Y 502.798,Z 181.858,A -85,B 0,C 180,E1 -5898.932,E2 -5898.932} C_VEL
LIN {X 0,Y 502.795,Z 181.85,A -85,B 0,C 180,E1 -5902.046,E2 -5902.046} C_VEL
LIN {X 0,Y 502.797,Z 181.856,A -85,B 0,C 180,E1 -5905.034,E2 -5905.034} C_VEL
LIN {X 0,Y 502.784,Z 181.852,A -85,B 0,C 180,E1 -5907.915,E2 -5907.915} C_VEL
LIN {X 0,Y 502.824,Z 181.853,A -85,B 0,C 180,E1 -5910.712,E2 -5910.712} C_VEL
LIN {X 0,Y 502.865,Z 181.843,A -85,B 0,C 180,E1 -5913.439,E2 -5913.439} C_VEL
LIN {X 0,Y 502.776,Z 181.855,A -85,B 0,C 180,E1 -5916.085,E2 -5916.085} C_VEL
LIN {X 0,Y 502.785,Z 181.858,A -85,B 0,C 180,E1 -5918.689,E2 -5918.689} C_VEL
LIN {X 0,Y 502.824,Z 181.848,A -85,B 0,C 180,E1 -5921.248,E2 -5921.248} C_VEL
LIN {X 0,Y 502.85,Z 181.851,A -85,B 0,C 180,E1 -5924.6,E2 -5924.6} C_VEL
LIN {X 0,Y 502.878,Z 181.844,A -85,B 0,C 180,E1 -5928.039,E2 -5928.039} C_VEL
LIN {X 0,Y 502.867,Z 181.844,A -85,B 0,C 180,E1 -5931.156,E2 -5931.156} C_VEL
LIN {X 0,Y 502.926,Z 181.842,A -85,B 0,C 180,E1 -5934.386,E2 -5934.386} C_VEL
LIN {X 0,Y 503.023,Z 181.827,A -85,B 0,C 180,E1 -5937.597,E2 -5937.597} C_VEL
LIN {X 0,Y 503.047,Z 182.017,A -85,B 0,C 180,E1 -5940,E2 -5940} C_VEL
LIN {X 0,Y 503.069,Z 198.88,A -85,B 0,C 180,E1 -5942.802,E2 -5942.802} C_VEL
LIN {X 0,Y 503.026,Z 215.337,A -85,B 0,C 180,E1 -5945.612,E2 -5945.612} C_VEL
LIN {X 0,Y 503.085,Z 225.727,A -85,B 0,C 180,E1 -5947.399,E2 -5947.399} C_VEL
LIN {X 0,Y 504.565,Z 235.201,A -85,B 0,C 180,E1 -5947.629,E2 -5947.629} C_VEL
LIN {X 0,Y 504.007,Z 306.414,A -85,B 0,C 180,E1 -5948.772,E2 -5948.772} C_VEL
LIN {X 0,Y 503.917,Z 318.154,A -85,B 0,C 180,E1 -5949.128,E2 -5949.128} C_VEL
LIN {X 0,Y 503.754,Z 329.367,A -85,B 0,C 180,E1 -5949.637,E2 -5949.637} C_VEL
LIN {X 0,Y 503.538,Z 339.346,A -85,B 0,C 180,E1 -5950.25,E2 -5950.25} C_VEL
LIN {X 0,Y 503.274,Z 349.612,A -85,B 0,C 180,E1 -5951.07,E2 -5951.07} C_VEL
LIN {X 0,Y 503.042,Z 359.048,A -85,B 0,C 180,E1 -5952.049,E2 -5952.049} C_VEL
LIN {X 0,Y 502.819,Z 365.763,A -85,B 0,C 180,E1 -5952.922,E2 -5952.922} C_VEL
LIN {X 0,Y 502.688,Z 372.112,A -85,B 0,C 180,E1 -5953.955,E2 -5953.955} C_VEL
LIN {X 0,Y 502.555,Z 376.682,A -85,B 0,C 180,E1 -5954.883,E2 -5954.883} C_VEL
LIN {X 0,Y 502.407,Z 380.397,A -85,B 0,C 180,E1 -5955.829,E2 -5955.829} C_VEL
LIN {X 0,Y 502.308,Z 384.021,A -85,B 0,C 180,E1 -5957.086,E2 -5957.086} C_VEL
LIN {X 0,Y 502.248,Z 385.683,A -85,B 0,C 180,E1 -5957.929,E2 -5957.929} C_VEL
LIN {X 0,Y 502.218,Z 386.757,A -85,B 0,C 180,E1 -5958.775,E2 -5958.775} C_VEL
LIN {X 0,Y 502.213,Z 387.294,A -85,B 0,C 180,E1 -5959.624,E2 -5959.624} C_VEL
LIN {X 0,Y 502.223,Z 387.255,A -85,B 0,C 180,E1 -5960.477,E2 -5960.477} C_VEL
LIN {X 0,Y 502.204,Z 386.642,A -85,B 0,C 180,E1 -5961.337,E2 -5961.337} C_VEL
LIN {X 0,Y 502.264,Z 384.799,A -85,B 0,C 180,E1 -5962.555,E2 -5962.555} C_VEL
LIN {X 0,Y 502.375,Z 381.196,A -85,B 0,C 180,E1 -5963.934,E2 -5963.934} C_VEL
LIN {X 0,Y 502.458,Z 378.014,A -85,B 0,C 180,E1 -5964.81,E2 -5964.81} C_VEL
LIN {X 0,Y 502.592,Z 372.997,A -85,B 0,C 180,E1 -5965.894,E2 -5965.894} C_VEL
LIN {X 0,Y 502.732,Z 366.231,A -85,B 0,C 180,E1 -5967.022,E2 -5967.022} C_VEL
LIN {X 0,Y 502.906,Z 359.526,A -85,B 0,C 180,E1 -5967.914,E2 -5967.914} C_VEL
LIN {X 0,Y 503.141,Z 351.159,A -85,B 0,C 180,E1 -5968.809,E2 -5968.809} C_VEL
LIN {X 0,Y 503.401,Z 341.92,A -85,B 0,C 180,E1 -5969.595,E2 -5969.595} C_VEL
LIN {X 0,Y 503.598,Z 331.636,A -85,B 0,C 180,E1 -5970.274,E2 -5970.274} C_VEL
LIN {X 0,Y 503.826,Z 321.496,A -85,B 0,C 180,E1 -5970.781,E2 -5970.781} C_VEL
LIN {X 0,Y 503.945,Z 309.743,A -85,B 0,C 180,E1 -5971.192,E2 -5971.192} C_VEL
LIN {X 0,Y 504.02,Z 297.687,A -85,B 0,C 180,E1 -5971.443,E2 -5971.443} C_VEL
LIN {X 0,Y 504.429,Z 235.789,A -85,B 0,C 180,E1 -5972.379,E2 -5972.379} C_VEL
LIN {X 0,Y 503.853,Z 232.573,A -85,B 0,C 180,E1 -5972.466,E2 -5972.466} C_VEL
LIN {X 0,Y 501.711,Z 228.7,A -85,B 0,C 180,E1 -5972.68,E2 -5972.68} C_VEL
LIN {X 0,Y 498.677,Z 225.058,A -85,B 0,C 180,E1 -5973.03,E2 -5973.03} C_VEL
LIN {X 0,Y 496.546,Z 222.246,A -85,B 0,C 180,E1 -5973.427,E2 -5973.427} C_VEL
LIN {X 0,Y 495.997,Z 220.382,A -85,B 0,C 180,E1 -5973.758,E2 -5973.758} C_VEL
LIN {X 0,Y 496.276,Z 203.625,A -85,B 0,C 180,E1 -5977.003,E2 -5977.003} C_VEL
LIN {X 0,Y 496.433,Z 187.586,A -85,B 0,C 180,E1 -5980.139,E2 -5980.139} C_VEL
LIN {X 0,Y 495.831,Z 182.791,A -85,B 0,C 180,E1 -5981.168,E2 -5981.168} C_VEL
LIN {X 0,Y 495.735,Z 182.732,A -85,B 0,C 180,E1 -5984.859,E2 -5984.859} C_VEL
LIN {X 0,Y 495.755,Z 182.729,A -85,B 0,C 180,E1 -5988.219,E2 -5988.219} C_VEL
LIN {X 0,Y 495.748,Z 182.732,A -85,B 0,C 180,E1 -5991.408,E2 -5991.408} C_VEL
LIN {X 0,Y 495.754,Z 182.727,A -85,B 0,C 180,E1 -5994.463,E2 -5994.463} C_VEL
LIN {X 0,Y 495.766,Z 182.731,A -85,B 0,C 180,E1 -5997.405,E2 -5997.405} C_VEL
LIN {X 0,Y 495.765,Z 182.726,A -85,B 0,C 180,E1 -6000.253,E2 -6000.253} C_VEL
LIN {X 0,Y 495.833,Z 182.722,A -85,B 0,C 180,E1 -6003.248,E2 -6003.248} C_VEL
LIN {X 0,Y 495.747,Z 182.733,A -85,B 0,C 180,E1 -6005.724,E2 -6005.724} C_VEL
LIN {X 0,Y 495.741,Z 182.728,A -85,B 0,C 180,E1 -6008.371,E2 -6008.371} C_VEL
LIN {X 0,Y 495.782,Z 182.726,A -85,B 0,C 180,E1 -6010.971,E2 -6010.971} C_VEL
LIN {X 0,Y 495.776,Z 182.73,A -85,B 0,C 180,E1 -6013.529,E2 -6013.529} C_VEL
LIN {X 0,Y 495.797,Z 182.722,A -85,B 0,C 180,E1 -6016.055,E2 -6016.055} C_VEL
LIN {X 0,Y 495.85,Z 182.716,A -85,B 0,C 180,E1 -6018.554,E2 -6018.554} C_VEL
LIN {X 0,Y 495.871,Z 182.713,A -85,B 0,C 180,E1 -6021.852,E2 -6021.852} C_VEL
LIN {X 0,Y 495.897,Z 182.709,A -85,B 0,C 180,E1 -6024.306,E2 -6024.306} C_VEL
LIN {X 0,Y 495.992,Z 182.7,A -85,B 0,C 180,E1 -6027.563,E2 -6027.563} C_VEL
LIN {X 0,Y 495.997,Z 182.697,A -85,B 0,C 180,E1 -6029.999,E2 -6029.999} C_VEL
LIN {X 0,Y 495.992,Z 182.699,A -85,B 0,C 180,E1 -6032.436,E2 -6032.436} C_VEL
LIN {X 0,Y 495.887,Z 182.711,A -85,B 0,C 180,E1 -6035.693,E2 -6035.693} C_VEL
LIN {X 0,Y 495.87,Z 182.713,A -85,B 0,C 180,E1 -6038.147,E2 -6038.147} C_VEL
LIN {X 0,Y 495.848,Z 182.717,A -85,B 0,C 180,E1 -6041.445,E2 -6041.445} C_VEL
LIN {X 0,Y 495.786,Z 182.731,A -85,B 0,C 180,E1 -6044.782,E2 -6044.782} C_VEL
LIN {X 0,Y 495.782,Z 182.725,A -85,B 0,C 180,E1 -6047.318,E2 -6047.318} C_VEL
LIN {X 0,Y 495.773,Z 182.724,A -85,B 0,C 180,E1 -6049.889,E2 -6049.889} C_VEL
LIN {X 0,Y 495.753,Z 182.734,A -85,B 0,C 180,E1 -6052.86,E2 -6052.86} C_VEL
LIN {X 0,Y 495.794,Z 182.723,A -85,B 0,C 180,E1 -6056.067,E2 -6056.067} C_VEL
LIN {X 0,Y 495.767,Z 182.731,A -85,B 0,C 180,E1 -6058.814,E2 -6058.814} C_VEL
LIN {X 0,Y 495.752,Z 182.727,A -85,B 0,C 180,E1 -6061.725,E2 -6061.725} C_VEL
LIN {X 0,Y 495.771,Z 182.731,A -85,B 0,C 180,E1 -6064.695,E2 -6064.695} C_VEL
LIN {X 0,Y 495.725,Z 182.73,A -85,B 0,C 180,E1 -6067.561,E2 -6067.561} C_VEL
LIN {X 0,Y 495.772,Z 182.73,A -85,B 0,C 180,E1 -6070.698,E2 -6070.698} C_VEL
LIN {X 0,Y 495.727,Z 182.731,A -85,B 0,C 180,E1 -6073.695,E2 -6073.695} C_VEL
LIN {X 0,Y 495.72,Z 182.739,A -85,B 0,C 180,E1 -6076.305,E2 -6076.305} C_VEL
LIN {X 0,Y 495.772,Z 182.725,A -85,B 0,C 180,E1 -6079.301,E2 -6079.301} C_VEL
LIN {X 0,Y 495.724,Z 182.737,A -85,B 0,C 180,E1 -6082.438,E2 -6082.438} C_VEL
LIN {X 0,Y 495.777,Z 182.724,A -85,B 0,C 180,E1 -6085.457,E2 -6085.457} C_VEL
LIN {X 0,Y 495.751,Z 182.733,A -85,B 0,C 180,E1 -6088.364,E2 -6088.364} C_VEL
LIN {X 0,Y 495.781,Z 182.725,A -85,B 0,C 180,E1 -6091.506,E2 -6091.506} C_VEL
LIN {X 0,Y 495.782,Z 182.73,A -85,B 0,C 180,E1 -6093.932,E2 -6093.932} C_VEL
LIN {X 0,Y 495.756,Z 182.727,A -85,B 0,C 180,E1 -6097.138,E2 -6097.138} C_VEL
LIN {X 0,Y 495.77,Z 182.732,A -85,B 0,C 180,E1 -6100.11,E2 -6100.11} C_VEL
LIN {X 0,Y 495.779,Z 182.724,A -85,B 0,C 180,E1 -6102.682,E2 -6102.682} C_VEL
LIN {X 0,Y 495.781,Z 182.724,A -85,B 0,C 180,E1 -6105.217,E2 -6105.217} C_VEL
LIN {X 0,Y 495.846,Z 182.716,A -85,B 0,C 180,E1 -6108.555,E2 -6108.555} C_VEL
LIN {X 0,Y 495.864,Z 182.721,A -85,B 0,C 180,E1 -6111.852,E2 -6111.852} C_VEL
LIN {X 0,Y 495.886,Z 182.712,A -85,B 0,C 180,E1 -6114.307,E2 -6114.307} C_VEL
LIN {X 0,Y 495.984,Z 182.705,A -85,B 0,C 180,E1 -6117.564,E2 -6117.564} C_VEL
LIN {X 0,Y 495.989,Z 182.702,A -85,B 0,C 180,E1 -6120,E2 -6120} C_VEL
LIN {X 0,Y 495.984,Z 182.698,A -85,B 0,C 180,E1 -6122.437,E2 -6122.437} C_VEL
LIN {X 0,Y 495.88,Z 182.718,A -85,B 0,C 180,E1 -6125.694,E2 -6125.694} C_VEL
LIN {X 0,Y 495.863,Z 182.715,A -85,B 0,C 180,E1 -6128.148,E2 -6128.148} C_VEL
LIN {X 0,Y 495.843,Z 182.724,A -85,B 0,C 180,E1 -6131.446,E2 -6131.446} C_VEL
LIN {X 0,Y 495.782,Z 182.724,A -85,B 0,C 180,E1 -6134.783,E2 -6134.783} C_VEL
LIN {X 0,Y 495.773,Z 182.732,A -85,B 0,C 180,E1 -6137.319,E2 -6137.319} C_VEL
LIN {X 0,Y 495.763,Z 182.728,A -85,B 0,C 180,E1 -6139.891,E2 -6139.891} C_VEL
LIN {X 0,Y 495.752,Z 182.73,A -85,B 0,C 180,E1 -6142.861,E2 -6142.861} C_VEL
LIN {X 0,Y 495.783,Z 182.723,A -85,B 0,C 180,E1 -6146.069,E2 -6146.069} C_VEL
LIN {X 0,Y 495.763,Z 182.729,A -85,B 0,C 180,E1 -6148.816,E2 -6148.816} C_VEL
LIN {X 0,Y 495.749,Z 182.729,A -85,B 0,C 180,E1 -6151.726,E2 -6151.726} C_VEL
LIN {X 0,Y 495.757,Z 182.729,A -85,B 0,C 180,E1 -6154.694,E2 -6154.694} C_VEL
LIN {X 0,Y 495.723,Z 182.733,A -85,B 0,C 180,E1 -6157.563,E2 -6157.563} C_VEL
LIN {X 0,Y 495.761,Z 182.73,A -85,B 0,C 180,E1 -6160.701,E2 -6160.701} C_VEL
LIN {X 0,Y 495.73,Z 182.73,A -85,B 0,C 180,E1 -6164.002,E2 -6164.002} C_VEL
LIN {X 0,Y 495.713,Z 182.738,A -85,B 0,C 180,E1 -6167.117,E2 -6167.117} C_VEL
LIN {X 0,Y 495.753,Z 182.729,A -85,B 0,C 180,E1 -6170.363,E2 -6170.363} C_VEL
LIN {X 0,Y 495.714,Z 182.733,A -85,B 0,C 180,E1 -6173.456,E2 -6173.456} C_VEL
LIN {X 0,Y 495.757,Z 182.732,A -85,B 0,C 180,E1 -6176.437,E2 -6176.437} C_VEL
LIN {X 0,Y 495.748,Z 182.733,A -85,B 0,C 180,E1 -6179.313,E2 -6179.313} C_VEL
LIN {X 0,Y 495.741,Z 182.734,A -85,B 0,C 180,E1 -6182.107,E2 -6182.107} C_VEL
LIN {X 0,Y 495.811,Z 182.892,A -85,B 0,C 180,E1 -6183.391,E2 -6183.391} C_VEL
LIN {X 0,Y 498.636,Z 195.539,A -85,B 0,C 180,E1 -6185.21,E2 -6185.21} C_VEL
LIN {X 0,Y 498.632,Z 200.654,A -85,B 0,C 180,E1 -6185.875,E2 -6185.875} C_VEL
LIN {X 0,Y 497.745,Z 225.378,A -85,B 0,C 180,E1 -6189.018,E2 -6189.018} C_VEL
LIN {X 0,Y 496.885,Z 253.272,A -85,B 0,C 180,E1 -6192.509,E2 -6192.509} C_VEL
LIN {X 0,Y 496.54,Z 266.699,A -85,B 0,C 180,E1 -6194.14,E2 -6194.14} C_VEL
LIN {X 0,Y 498.101,Z 281.58,A -85,B 0,C 180,E1 -6194.422,E2 -6194.422} C_VEL
LIN {X 0,Y 497.513,Z 375.147,A -85,B 0,C 180,E1 -6195.819,E2 -6195.819} C_VEL
LIN {X 0,Y 497.278,Z 388.418,A -85,B 0,C 180,E1 -6196.177,E2 -6196.177} C_VEL
LIN {X 0,Y 496.953,Z 400.583,A -85,B 0,C 180,E1 -6196.663,E2 -6196.663} C_VEL
LIN {X 0,Y 496.588,Z 412.842,A -85,B 0,C 180,E1 -6197.329,E2 -6197.329} C_VEL
LIN {X 0,Y 496.292,Z 424.465,A -85,B 0,C 180,E1 -6198.152,E2 -6198.152} C_VEL
LIN {X 0,Y 495.955,Z 433.838,A -85,B 0,C 180,E1 -6198.972,E2 -6198.972} C_VEL
LIN {X 0,Y 495.664,Z 443.452,A -85,B 0,C 180,E1 -6199.998,E2 -6199.998} C_VEL
LIN {X 0,Y 495.405,Z 452.686,A -85,B 0,C 180,E1 -6201.229,E2 -6201.229} C_VEL
LIN {X 0,Y 495.243,Z 460.116,A -85,B 0,C 180,E1 -6202.458,E2 -6202.458} C_VEL
LIN {X 0,Y 495.133,Z 466.356,A -85,B 0,C 180,E1 -6203.754,E2 -6203.754} C_VEL
LIN {X 0,Y 495.047,Z 471.368,A -85,B 0,C 180,E1 -6205.114,E2 -6205.114} C_VEL
LIN {X 0,Y 495.167,Z 473.733,A -85,B 0,C 180,E1 -6205.931,E2 -6205.931} C_VEL
LIN {X 0,Y 495.204,Z 475.65,A -85,B 0,C 180,E1 -6206.746,E2 -6206.746} C_VEL
LIN {X 0,Y 495.075,Z 477.078,A -85,B 0,C 180,E1 -6207.56,E2 -6207.56} C_VEL
LIN {X 0,Y 495.014,Z 478.696,A -85,B 0,C 180,E1 -6209.187,E2 -6209.187} C_VEL
LIN {X 0,Y 495.025,Z 478.906,A -85,B 0,C 180,E1 -6210.001,E2 -6210.001} C_VEL
LIN {X 0,Y 495.017,Z 478.666,A -85,B 0,C 180,E1 -6210.814,E2 -6210.814} C_VEL
LIN {X 0,Y 495.077,Z 476.977,A -85,B 0,C 180,E1 -6212.441,E2 -6212.441} C_VEL
LIN {X 0,Y 495.204,Z 475.519,A -85,B 0,C 180,E1 -6213.255,E2 -6213.255} C_VEL
LIN {X 0,Y 495.111,Z 472.443,A -85,B 0,C 180,E1 -6214.478,E2 -6214.478} C_VEL
LIN {X 0,Y 495.162,Z 467.187,A -85,B 0,C 180,E1 -6215.976,E2 -6215.976} C_VEL
LIN {X 0,Y 495.261,Z 460.873,A -85,B 0,C 180,E1 -6217.338,E2 -6217.338} C_VEL
LIN {X 0,Y 495.363,Z 453.645,A -85,B 0,C 180,E1 -6218.568,E2 -6218.568} C_VEL
LIN {X 0,Y 495.549,Z 444.602,A -85,B 0,C 180,E1 -6219.799,E2 -6219.799} C_VEL
LIN {X 0,Y 495.878,Z 435.338,A -85,B 0,C 180,E1 -6220.824,E2 -6220.824} C_VEL
LIN {X 0,Y 496.188,Z 425.152,A -85,B 0,C 180,E1 -6221.742,E2 -6221.742} C_VEL
LIN {X 0,Y 496.497,Z 413.786,A -85,B 0,C 180,E1 -6222.56,E2 -6222.56} C_VEL
LIN {X 0,Y 496.861,Z 401.755,A -85,B 0,C 180,E1 -6223.237,E2 -6223.237} C_VEL
LIN {X 0,Y 497.207,Z 388.749,A -85,B 0,C 180,E1 -6223.774,E2 -6223.774} C_VEL
LIN {X 0,Y 497.507,Z 374.8,A -85,B 0,C 180,E1 -6224.156,E2 -6224.156} C_VEL
LIN {X 0,Y 497.955,Z 279.082,A -85,B 0,C 180,E1 -6225.606,E2 -6225.606} C_VEL
LIN {X 0,Y 496.446,Z 265.697,A -85,B 0,C 180,E1 -6225.879,E2 -6225.879} C_VEL
LIN {X 0,Y 497.035,Z 241.819,A -85,B 0,C 180,E1 -6228.75,E2 -6228.75} C_VEL
LIN {X 0,Y 497.737,Z 215.346,A -85,B 0,C 180,E1 -6231.974,E2 -6231.974} C_VEL
LIN {X 0,Y 498.28,Z 195.95,A -85,B 0,C 180,E1 -6234.366,E2 -6234.366} C_VEL
LIN {X 0,Y 497.872,Z 192.372,A -85,B 0,C 180,E1 -6234.832,E2 -6234.832} C_VEL
LIN {X 0,Y 495.797,Z 182.86,A -85,B 0,C 180,E1 -6236.167,E2 -6236.167} C_VEL
LIN {X 0,Y 495.761,Z 182.733,A -85,B 0,C 180,E1 -6239.747,E2 -6239.747} C_VEL
LIN {X 0,Y 495.769,Z 182.73,A -85,B 0,C 180,E1 -6242.595,E2 -6242.595} C_VEL
LIN {X 0,Y 495.747,Z 182.734,A -85,B 0,C 180,E1 -6245.538,E2 -6245.538} C_VEL
LIN {X 0,Y 495.761,Z 182.731,A -85,B 0,C 180,E1 -6248.767,E2 -6248.767} C_VEL
LIN {X 0,Y 495.746,Z 182.731,A -85,B 0,C 180,E1 -6251.782,E2 -6251.782} C_VEL
LIN {X 0,Y 495.74,Z 182.736,A -85,B 0,C 180,E1 -6255.141,E2 -6255.141} C_VEL
LIN {X 0,Y 495.752,Z 182.728,A -85,B 0,C 180,E1 -6258.218,E2 -6258.218} C_VEL
LIN {X 0,Y 495.751,Z 182.73,A -85,B 0,C 180,E1 -6261.408,E2 -6261.408} C_VEL
LIN {X 0,Y 495.749,Z 182.732,A -85,B 0,C 180,E1 -6264.462,E2 -6264.462} C_VEL
LIN {X 0,Y 495.768,Z 182.728,A -85,B 0,C 180,E1 -6267.405,E2 -6267.405} C_VEL
LIN {X 0,Y 495.767,Z 182.729,A -85,B 0,C 180,E1 -6270.253,E2 -6270.253} C_VEL
LIN {X 0,Y 495.825,Z 182.721,A -85,B 0,C 180,E1 -6273.251,E2 -6273.251} C_VEL
LIN {X 0,Y 495.744,Z 182.735,A -85,B 0,C 180,E1 -6276.612,E2 -6276.612} C_VEL
LIN {X 0,Y 495.78,Z 182.725,A -85,B 0,C 180,E1 -6279.324,E2 -6279.324} C_VEL
LIN {X 0,Y 495.78,Z 182.726,A -85,B 0,C 180,E1 -6281.828,E2 -6281.828} C_VEL
LIN {X 0,Y 495.825,Z 182.725,A -85,B 0,C 180,E1 -6284.548,E2 -6284.548} C_VEL
LIN {X 0,Y 495.83,Z 182.721,A -85,B 0,C 180,E1 -6287.965,E2 -6287.965} C_VEL
LIN {X 0,Y 495.838,Z 182.72,A -85,B 0,C 180,E1 -6291.03,E2 -6291.03} C_VEL
LIN {X 0,Y 495.881,Z 182.719,A -85,B 0,C 180,E1 -6294.306,E2 -6294.306} C_VEL
LIN {X 0,Y 495.992,Z 182.703,A -85,B 0,C 180,E1 -6297.563,E2 -6297.563} C_VEL
LIN {X 0,Y 495.994,Z 182.847,A -85,B 0,C 180,E1 -6299.847,E2 -6299.847} C_VEL
LIN {X 0,Y 496.096,Z 195.828,A -85,B 0,C 180,E1 -6302.029,E2 -6302.029} C_VEL
LIN {X 0,Y 496.096,Z 213.795,A -85,B 0,C 180,E1 -6305.079,E2 -6305.079} C_VEL
LIN {X 0,Y 496.073,Z 225.949,A -85,B 0,C 180,E1 -6307.176,E2 -6307.176} C_VEL
LIN {X 0,Y 496.979,Z 231.033,A -85,B 0,C 180,E1 -6307.326,E2 -6307.326} C_VEL
LIN {X 0,Y 497.699,Z 236.096,A -85,B 0,C 180,E1 -6307.434,E2 -6307.434} C_VEL
LIN {X 0,Y 497.106,Z 305.964,A -85,B 0,C 180,E1 -6308.58,E2 -6308.58} C_VEL
LIN {X 0,Y 496.99,Z 318.299,A -85,B 0,C 180,E1 -6308.948,E2 -6308.948} C_VEL
LIN {X 0,Y 496.809,Z 329.614,A -85,B 0,C 180,E1 -6309.465,E2 -6309.465} C_VEL
LIN {X 0,Y 496.59,Z 339.685,A -85,B 0,C 180,E1 -6310.086,E2 -6310.086} C_VEL
LIN {X 0,Y 496.325,Z 350.005,A -85,B 0,C 180,E1 -6310.917,E2 -6310.917} C_VEL
LIN {X 0,Y 496.105,Z 358.079,A -85,B 0,C 180,E1 -6311.746,E2 -6311.746} C_VEL
LIN {X 0,Y 495.868,Z 365.513,A -85,B 0,C 180,E1 -6312.69,E2 -6312.69} C_VEL
LIN {X 0,Y 495.69,Z 372.074,A -85,B 0,C 180,E1 -6313.738,E2 -6313.738} C_VEL
LIN {X 0,Y 495.481,Z 378.328,A -85,B 0,C 180,E1 -6315.035,E2 -6315.035} C_VEL
LIN {X 0,Y 495.355,Z 382.026,A -85,B 0,C 180,E1 -6316.061,E2 -6316.061} C_VEL
LIN {X 0,Y 495.247,Z 385.32,A -85,B 0,C 180,E1 -6317.338,E2 -6317.338} C_VEL
LIN {X 0,Y 495.167,Z 386.775,A -85,B 0,C 180,E1 -6318.194,E2 -6318.194} C_VEL
LIN {X 0,Y 495.165,Z 387.677,A -85,B 0,C 180,E1 -6319.053,E2 -6319.053} C_VEL
LIN {X 0,Y 495.153,Z 387.905,A -85,B 0,C 180,E1 -6320.483,E2 -6320.483} C_VEL
LIN {X 0,Y 495.158,Z 386.954,A -85,B 0,C 180,E1 -6321.655,E2 -6321.655} C_VEL
LIN {X 0,Y 495.216,Z 385.18,A -85,B 0,C 180,E1 -6322.711,E2 -6322.711} C_VEL
LIN {X 0,Y 495.329,Z 382.232,A -85,B 0,C 180,E1 -6323.851,E2 -6323.851} C_VEL
LIN {X 0,Y 495.441,Z 377.335,A -85,B 0,C 180,E1 -6325.186,E2 -6325.186} C_VEL
LIN {X 0,Y 495.602,Z 371.313,A -85,B 0,C 180,E1 -6326.391,E2 -6326.391} C_VEL
LIN {X 0,Y 495.792,Z 364.624,A -85,B 0,C 180,E1 -6327.432,E2 -6327.432} C_VEL
LIN {X 0,Y 496.013,Z 356.303,A -85,B 0,C 180,E1 -6328.459,E2 -6328.459} C_VEL
LIN {X 0,Y 496.27,Z 346.936,A -85,B 0,C 180,E1 -6329.363,E2 -6329.363} C_VEL
LIN {X 0,Y 496.546,Z 337.592,A -85,B 0,C 180,E1 -6330.075,E2 -6330.075} C_VEL
LIN {X 0,Y 496.769,Z 326.209,A -85,B 0,C 180,E1 -6330.735,E2 -6330.735} C_VEL
LIN {X 0,Y 496.949,Z 314.649,A -85,B 0,C 180,E1 -6331.21,E2 -6331.21} C_VEL
LIN {X 0,Y 497.03,Z 303.241,A -85,B 0,C 180,E1 -6331.516,E2 -6331.516} C_VEL
LIN {X 0,Y 497.435,Z 234.421,A -85,B 0,C 180,E1 -6332.588,E2 -6332.588} C_VEL
LIN {X 0,Y 495.946,Z 225.642,A -85,B 0,C 180,E1 -6332.799,E2 -6332.799} C_VEL
LIN {X 0,Y 495.997,Z 220.382,A -85,B 0,C 180,E1 -6333.758,E2 -6333.758} C_VEL
LIN {X 0,Y 495.429,Z 217.461,A -85,B 0,C 180,E1 -6334.347,E2 -6334.347} C_VEL
LIN {X 0,Y 492.657,Z 212.953,A -85,B 0,C 180,E1 -6335.32,E2 -6335.32} C_VEL
LIN {X 0,Y 489.854,Z 208.437,A -85,B 0,C 180,E1 -6336.304,E2 -6336.304} C_VEL
LIN {X 0,Y 489.247,Z 205.485,A -85,B 0,C 180,E1 -6336.902,E2 -6336.902} C_VEL
LIN {X 0,Y 489.452,Z 189.826,A -85,B 0,C 180,E1 -6339.982,E2 -6339.982} C_VEL
LIN {X 0,Y 489.025,Z 185.021,A -85,B 0,C 180,E1 -6340.953,E2 -6340.953} C_VEL
LIN {X 0,Y 488.78,Z 183.619,A -85,B 0,C 180,E1 -6341.338,E2 -6341.338} C_VEL
LIN {X 0,Y 488.7,Z 183.609,A -85,B 0,C 180,E1 -6344.802,E2 -6344.802} C_VEL
LIN {X 0,Y 488.69,Z 183.614,A -85,B 0,C 180,E1 -6347.474,E2 -6347.474} C_VEL
LIN {X 0,Y 488.731,Z 183.61,A -85,B 0,C 180,E1 -6349.676,E2 -6349.676} C_VEL
LIN {X 0,Y 488.68,Z 183.608,A -85,B 0,C 180,E1 -6352.841,E2 -6352.841} C_VEL
LIN {X 0,Y 488.732,Z 183.606,A -85,B 0,C 180,E1 -6355.887,E2 -6355.887} C_VEL
LIN {X 0,Y 488.69,Z 183.607,A -85,B 0,C 180,E1 -6358.82,E2 -6358.82} C_VEL
LIN {X 0,Y 488.744,Z 183.607,A -85,B 0,C 180,E1 -6361.671,E2 -6361.671} C_VEL
LIN {X 0,Y 488.749,Z 183.599,A -85,B 0,C 180,E1 -6364.444,E2 -6364.444} C_VEL
LIN {X 0,Y 488.721,Z 183.607,A -85,B 0,C 180,E1 -6367.153,E2 -6367.153} C_VEL
LIN {X 0,Y 488.723,Z 183.606,A -85,B 0,C 180,E1 -6369.81,E2 -6369.81} C_VEL
LIN {X 0,Y 488.728,Z 183.602,A -85,B 0,C 180,E1 -6372.423,E2 -6372.423} C_VEL
LIN {X 0,Y 488.763,Z 183.602,A -85,B 0,C 180,E1 -6374.999,E2 -6374.999} C_VEL
LIN {X 0,Y 488.804,Z 183.593,A -85,B 0,C 180,E1 -6378.387,E2 -6378.387} C_VEL
LIN {X 0,Y 488.816,Z 183.593,A -85,B 0,C 180,E1 -6381.733,E2 -6381.733} C_VEL
LIN {X 0,Y 488.856,Z 183.586,A -85,B 0,C 180,E1 -6384.224,E2 -6384.224} C_VEL
LIN {X 0,Y 488.96,Z 183.576,A -85,B 0,C 180,E1 -6387.528,E2 -6387.528} C_VEL
LIN {X 0,Y 488.952,Z 183.579,A -85,B 0,C 180,E1 -6390.823,E2 -6390.823} C_VEL
LIN {X 0,Y 488.959,Z 183.575,A -85,B 0,C 180,E1 -6392.471,E2 -6392.471} C_VEL
LIN {X 0,Y 488.845,Z 183.588,A -85,B 0,C 180,E1 -6395.775,E2 -6395.775} C_VEL
LIN {X 0,Y 488.814,Z 183.592,A -85,B 0,C 180,E1 -6398.266,E2 -6398.266} C_VEL
LIN {X 0,Y 488.802,Z 183.593,A -85,B 0,C 180,E1 -6401.612,E2 -6401.612} C_VEL
LIN {X 0,Y 488.758,Z 183.605,A -85,B 0,C 180,E1 -6405,E2 -6405} C_VEL
LIN {X 0,Y 488.75,Z 183.603,A -85,B 0,C 180,E1 -6408.441,E2 -6408.441} C_VEL
LIN {X 0,Y 488.703,Z 183.609,A -85,B 0,C 180,E1 -6411.07,E2 -6411.07} C_VEL
LIN {X 0,Y 488.689,Z 183.607,A -85,B 0,C 180,E1 -6413.745,E2 -6413.745} C_VEL
LIN {X 0,Y 488.793,Z 183.598,A -85,B 0,C 180,E1 -6416.945,E2 -6416.945} C_VEL
LIN {X 0,Y 488.704,Z 183.61,A -85,B 0,C 180,E1 -6420.362,E2 -6420.362} C_VEL
LIN {X 0,Y 488.73,Z 183.602,A -85,B 0,C 180,E1 -6423.484,E2 -6423.484} C_VEL
LIN {X 0,Y 488.683,Z 183.614,A -85,B 0,C 180,E1 -6426.355,E2 -6426.355} C_VEL
LIN {X 0,Y 488.735,Z 183.602,A -85,B 0,C 180,E1 -6429.25,E2 -6429.25} C_VEL
LIN {X 0,Y 488.724,Z 183.61,A -85,B 0,C 180,E1 -6432.521,E2 -6432.521} C_VEL
LIN {X 0,Y 488.704,Z 183.605,A -85,B 0,C 180,E1 -6435.198,E2 -6435.198} C_VEL
LIN {X 0,Y 488.704,Z 183.613,A -85,B 0,C 180,E1 -6438.399,E2 -6438.399} C_VEL
LIN {X 0,Y 488.732,Z 183.602,A -85,B 0,C 180,E1 -6440.942,E2 -6440.942} C_VEL
LIN {X 0,Y 488.677,Z 183.612,A -85,B 0,C 180,E1 -6443.868,E2 -6443.868} C_VEL
LIN {X 0,Y 488.731,Z 183.603,A -85,B 0,C 180,E1 -6446.877,E2 -6446.877} C_VEL
LIN {X 0,Y 488.726,Z 183.606,A -85,B 0,C 180,E1 -6449.781,E2 -6449.781} C_VEL
LIN {X 0,Y 488.783,Z 183.595,A -85,B 0,C 180,E1 -6453.056,E2 -6453.056} C_VEL
LIN {X 0,Y 488.685,Z 183.613,A -85,B 0,C 180,E1 -6456.255,E2 -6456.255} C_VEL
LIN {X 0,Y 488.737,Z 183.601,A -85,B 0,C 180,E1 -6459.176,E2 -6459.176} C_VEL
LIN {X 0,Y 488.75,Z 183.603,A -85,B 0,C 180,E1 -6461.628,E2 -6461.628} C_VEL
LIN {X 0,Y 488.753,Z 183.599,A -85,B 0,C 180,E1 -6465,E2 -6465} C_VEL
LIN {X 0,Y 488.799,Z 183.595,A -85,B 0,C 180,E1 -6468.388,E2 -6468.388} C_VEL
LIN {X 0,Y 488.809,Z 183.6,A -85,B 0,C 180,E1 -6471.734,E2 -6471.734} C_VEL
LIN {X 0,Y 488.846,Z 183.59,A -85,B 0,C 180,E1 -6474.225,E2 -6474.225} C_VEL
LIN {X 0,Y 488.952,Z 183.58,A -85,B 0,C 180,E1 -6477.529,E2 -6477.529} C_VEL
LIN {X 0,Y 488.946,Z 183.575,A -85,B 0,C 180,E1 -6480.824,E2 -6480.824} C_VEL
LIN {X 0,Y 488.952,Z 183.574,A -85,B 0,C 180,E1 -6482.472,E2 -6482.472} C_VEL
LIN {X 0,Y 488.839,Z 183.594,A -85,B 0,C 180,E1 -6485.776,E2 -6485.776} C_VEL
LIN {X 0,Y 488.808,Z 183.593,A -85,B 0,C 180,E1 -6488.267,E2 -6488.267} C_VEL
LIN {X 0,Y 488.797,Z 183.6,A -85,B 0,C 180,E1 -6491.613,E2 -6491.613} C_VEL
LIN {X 0,Y 488.754,Z 183.602,A -85,B 0,C 180,E1 -6495.001,E2 -6495.001} C_VEL
LIN {X 0,Y 488.748,Z 183.6,A -85,B 0,C 180,E1 -6498.443,E2 -6498.443} C_VEL
LIN {X 0,Y 488.7,Z 183.61,A -85,B 0,C 180,E1 -6501.071,E2 -6501.071} C_VEL
LIN {X 0,Y 488.677,Z 183.611,A -85,B 0,C 180,E1 -6503.747,E2 -6503.747} C_VEL
LIN {X 0,Y 488.785,Z 183.599,A -85,B 0,C 180,E1 -6506.944,E2 -6506.944} C_VEL
LIN {X 0,Y 488.703,Z 183.605,A -85,B 0,C 180,E1 -6510.364,E2 -6510.364} C_VEL
LIN {X 0,Y 488.723,Z 183.607,A -85,B 0,C 180,E1 -6513.484,E2 -6513.484} C_VEL
LIN {X 0,Y 488.677,Z 183.609,A -85,B 0,C 180,E1 -6516.355,E2 -6516.355} C_VEL
LIN {X 0,Y 488.696,Z 183.612,A -85,B 0,C 180,E1 -6519.255,E2 -6519.255} C_VEL
LIN {X 0,Y 488.702,Z 183.607,A -85,B 0,C 180,E1 -6521.601,E2 -6521.601} C_VEL
LIN {X 0,Y 488.708,Z 183.611,A -85,B 0,C 180,E1 -6524.802,E2 -6524.802} C_VEL
LIN {X 0,Y 488.684,Z 183.609,A -85,B 0,C 180,E1 -6527.475,E2 -6527.475} C_VEL
LIN {X 0,Y 488.698,Z 183.612,A -85,B 0,C 180,E1 -6530.747,E2 -6530.747} C_VEL
LIN {X 0,Y 488.667,Z 183.61,A -85,B 0,C 180,E1 -6533.868,E2 -6533.868} C_VEL
LIN {X 0,Y 488.737,Z 183.609,A -85,B 0,C 180,E1 -6536.878,E2 -6536.878} C_VEL
LIN {X 0,Y 488.72,Z 183.607,A -85,B 0,C 180,E1 -6539.782,E2 -6539.782} C_VEL
LIN {X 0,Y 488.754,Z 183.739,A -85,B 0,C 180,E1 -6543.154,E2 -6543.154} C_VEL
LIN {X 0,Y 491.931,Z 198.488,A -85,B 0,C 180,E1 -6545.3,E2 -6545.3} C_VEL
LIN {X 0,Y 490.889,Z 224.458,A -85,B 0,C 180,E1 -6548.652,E2 -6548.652} C_VEL
LIN {X 0,Y 489.956,Z 251.064,A -85,B 0,C 180,E1 -6552.038,E2 -6552.038} C_VEL
LIN {X 0,Y 489.526,Z 266.212,A -85,B 0,C 180,E1 -6553.924,E2 -6553.924} C_VEL
LIN {X 0,Y 491.22,Z 281.302,A -85,B 0,C 180,E1 -6554.227,E2 -6554.227} C_VEL
LIN {X 0,Y 490.591,Z 374.577,A -85,B 0,C 180,E1 -6555.641,E2 -6555.641} C_VEL
LIN {X 0,Y 490.332,Z 387.865,A -85,B 0,C 180,E1 -6556.004,E2 -6556.004} C_VEL
LIN {X 0,Y 489.966,Z 400.603,A -85,B 0,C 180,E1 -6556.522,E2 -6556.522} C_VEL
LIN {X 0,Y 489.599,Z 411.892,A -85,B 0,C 180,E1 -6557.145,E2 -6557.145} C_VEL
LIN {X 0,Y 489.363,Z 422.158,A -85,B 0,C 180,E1 -6557.866,E2 -6557.866} C_VEL
LIN {X 0,Y 488.869,Z 433.013,A -85,B 0,C 180,E1 -6558.81,E2 -6558.81} C_VEL
LIN {X 0,Y 488.589,Z 442.683,A -85,B 0,C 180,E1 -6559.852,E2 -6559.852} C_VEL
LIN {X 0,Y 488.34,Z 451.962,A -85,B 0,C 180,E1 -6561.101,E2 -6561.101} C_VEL
LIN {X 0,Y 488.177,Z 459.418,A -85,B 0,C 180,E1 -6562.348,E2 -6562.348} C_VEL
LIN {X 0,Y 488.096,Z 464.86,A -85,B 0,C 180,E1 -6563.475,E2 -6563.475} C_VEL
LIN {X 0,Y 488.056,Z 469.347,A -85,B 0,C 180,E1 -6564.63,E2 -6564.63} C_VEL
LIN {X 0,Y 488.076,Z 473.078,A -85,B 0,C 180,E1 -6565.872,E2 -6565.872} C_VEL
LIN {X 0,Y 488.117,Z 474.999,A -85,B 0,C 180,E1 -6566.699,E2 -6566.699} C_VEL
LIN {X 0,Y 488.014,Z 476.433,A -85,B 0,C 180,E1 -6567.524,E2 -6567.524} C_VEL
LIN {X 0,Y 487.942,Z 478.051,A -85,B 0,C 180,E1 -6569.175,E2 -6569.175} C_VEL
LIN {X 0,Y 487.955,Z 478.259,A -85,B 0,C 180,E1 -6570.001,E2 -6570.001} C_VEL
LIN {X 0,Y 487.945,Z 478.014,A -85,B 0,C 180,E1 -6570.826,E2 -6570.826} C_VEL
LIN {X 0,Y 488.016,Z 476.318,A -85,B 0,C 180,E1 -6572.477,E2 -6572.477} C_VEL
LIN {X 0,Y 488.131,Z 474.849,A -85,B 0,C 180,E1 -6573.302,E2 -6573.302} C_VEL
LIN {X 0,Y 488.011,Z 471.758,A -85,B 0,C 180,E1 -6574.544,E2 -6574.544} C_VEL
LIN {X 0,Y 488.088,Z 467.597,A -85,B 0,C 180,E1 -6575.785,E2 -6575.785} C_VEL
LIN {X 0,Y 488.179,Z 461.189,A -85,B 0,C 180,E1 -6577.237,E2 -6577.237} C_VEL
LIN {X 0,Y 488.277,Z 454.199,A -85,B 0,C 180,E1 -6578.484,E2 -6578.484} C_VEL
LIN {X 0,Y 488.42,Z 447.064,A -85,B 0,C 180,E1 -6579.525,E2 -6579.525} C_VEL
LIN {X 0,Y 488.711,Z 438.474,A -85,B 0,C 180,E1 -6580.566,E2 -6580.566} C_VEL
LIN {X 0,Y 489.024,Z 427.844,A -85,B 0,C 180,E1 -6581.608,E2 -6581.608} C_VEL
LIN {X 0,Y 489.314,Z 417.305,A -85,B 0,C 180,E1 -6582.442,E2 -6582.442} C_VEL
LIN {X 0,Y 489.71,Z 405.743,A -85,B 0,C 180,E1 -6583.17,E2 -6583.17} C_VEL
LIN {X 0,Y 490.121,Z 393.773,A -85,B 0,C 180,E1 -6583.739,E2 -6583.739} C_VEL
LIN {X 0,Y 490.449,Z 380.821,A -85,B 0,C 180,E1 -6584.179,E2 -6584.179} C_VEL
LIN {X 0,Y 490.666,Z 367.119,A -85,B 0,C 180,E1 -6584.464,E2 -6584.464} C_VEL
LIN {X 0,Y 491.1,Z 280.077,A -85,B 0,C 180,E1 -6585.79,E2 -6585.79} C_VEL
LIN {X 0,Y 489.455,Z 265.417,A -85,B 0,C 180,E1 -6586.092,E2 -6586.092} C_VEL
LIN {X 0,Y 490.09,Z 241.795,A -85,B 0,C 180,E1 -6588.968,E2 -6588.968} C_VEL
LIN {X 0,Y 490.828,Z 214.891,A -85,B 0,C 180,E1 -6592.3,E2 -6592.3} C_VEL
LIN {X 0,Y 491.404,Z 197.241,A -85,B 0,C 180,E1 -6594.504,E2 -6594.504} C_VEL
LIN {X 0,Y 490.159,Z 190.051,A -85,B 0,C 180,E1 -6595.477,E2 -6595.477} C_VEL
LIN {X 0,Y 488.761,Z 183.738,A -85,B 0,C 180,E1 -6596.4,E2 -6596.4} C_VEL
LIN {X 0,Y 488.704,Z 183.613,A -85,B 0,C 180,E1 -6599.272,E2 -6599.272} C_VEL
LIN {X 0,Y 488.705,Z 183.609,A -85,B 0,C 180,E1 -6602.147,E2 -6602.147} C_VEL
LIN {X 0,Y 488.716,Z 183.612,A -85,B 0,C 180,E1 -6605.115,E2 -6605.115} C_VEL
LIN {X 0,Y 488.677,Z 183.61,A -85,B 0,C 180,E1 -6608.201,E2 -6608.201} C_VEL
LIN {X 0,Y 488.696,Z 183.609,A -85,B 0,C 180,E1 -6610.341,E2 -6610.341} C_VEL
LIN {X 0,Y 488.679,Z 183.611,A -85,B 0,C 180,E1 -6613.656,E2 -6613.656} C_VEL
LIN {X 0,Y 488.679,Z 183.61,A -85,B 0,C 180,E1 -6616.344,E2 -6616.344} C_VEL
LIN {X 0,Y 488.706,Z 183.606,A -85,B 0,C 180,E1 -6619.673,E2 -6619.673} C_VEL
LIN {X 0,Y 488.681,Z 183.615,A -85,B 0,C 180,E1 -6622.841,E2 -6622.841} C_VEL
LIN {X 0,Y 488.726,Z 183.604,A -85,B 0,C 180,E1 -6625.886,E2 -6625.886} C_VEL
LIN {X 0,Y 488.693,Z 183.613,A -85,B 0,C 180,E1 -6628.82,E2 -6628.82} C_VEL
LIN {X 0,Y 488.744,Z 183.602,A -85,B 0,C 180,E1 -6631.671,E2 -6631.671} C_VEL
LIN {X 0,Y 488.754,Z 183.601,A -85,B 0,C 180,E1 -6633.528,E2 -6633.528} C_VEL
LIN {X 0,Y 488.678,Z 183.613,A -85,B 0,C 180,E1 -6636.253,E2 -6636.253} C_VEL
LIN {X 0,Y 488.748,Z 183.602,A -85,B 0,C 180,E1 -6639.175,E2 -6639.175} C_VEL
LIN {X 0,Y 488.749,Z 183.601,A -85,B 0,C 180,E1 -6641.632,E2 -6641.632} C_VEL
LIN {X 0,Y 488.763,Z 183.602,A -85,B 0,C 180,E1 -6644.999,E2 -6644.999} C_VEL
LIN {X 0,Y 488.807,Z 183.601,A -85,B 0,C 180,E1 -6648.387,E2 -6648.387} C_VEL
LIN {X 0,Y 488.787,Z 183.599,A -85,B 0,C 180,E1 -6651.733,E2 -6651.733} C_VEL
LIN {X 0,Y 488.838,Z 183.596,A -85,B 0,C 180,E1 -6654.224,E2 -6654.224} C_VEL
LIN {X 0,Y 488.96,Z 183.579,A -85,B 0,C 180,E1 -6657.528,E2 -6657.528} C_VEL
LIN {X 0,Y 488.966,Z 183.735,A -85,B 0,C 180,E1 -6659.691,E2 -6659.691} C_VEL
LIN {X 0,Y 489.183,Z 189.199,A -85,B 0,C 180,E1 -6660.617,E2 -6660.617} C_VEL
LIN {X 0,Y 489.111,Z 206.272,A -85,B 0,C 180,E1 -6663.501,E2 -6663.501} C_VEL
LIN {X 0,Y 489.09,Z 221.711,A -85,B 0,C 180,E1 -6666.186,E2 -6666.186} C_VEL
LIN {X 0,Y 489.141,Z 226.545,A -85,B 0,C 180,E1 -6666.978,E2 -6666.978} C_VEL
LIN {X 0,Y 490.855,Z 236.208,A -85,B 0,C 180,E1 -6667.217,E2 -6667.217} C_VEL
LIN {X 0,Y 490.194,Z 307.325,A -85,B 0,C 180,E1 -6668.423,E2 -6668.423} C_VEL
LIN {X 0,Y 490.078,Z 318.452,A -85,B 0,C 180,E1 -6668.763,E2 -6668.763} C_VEL
LIN {X 0,Y 489.889,Z 329.863,A -85,B 0,C 180,E1 -6669.287,E2 -6669.287} C_VEL
LIN {X 0,Y 489.666,Z 340.011,A -85,B 0,C 180,E1 -6669.917,E2 -6669.917} C_VEL
LIN {X 0,Y 489.382,Z 350.39,A -85,B 0,C 180,E1 -6670.759,E2 -6670.759} C_VEL
LIN {X 0,Y 489.137,Z 358.555,A -85,B 0,C 180,E1 -6671.604,E2 -6671.604} C_VEL
LIN {X 0,Y 488.85,Z 366.749,A -85,B 0,C 180,E1 -6672.664,E2 -6672.664} C_VEL
LIN {X 0,Y 488.672,Z 373.173,A -85,B 0,C 180,E1 -6673.727,E2 -6673.727} C_VEL
LIN {X 0,Y 488.444,Z 379.183,A -85,B 0,C 180,E1 -6675.01,E2 -6675.01} C_VEL
LIN {X 0,Y 488.319,Z 383.57,A -85,B 0,C 180,E1 -6676.298,E2 -6676.298} C_VEL
LIN {X 0,Y 488.167,Z 386.552,A -85,B 0,C 180,E1 -6677.597,E2 -6677.597} C_VEL
LIN {X 0,Y 488.105,Z 387.826,A -85,B 0,C 180,E1 -6678.467,E2 -6678.467} C_VEL
LIN {X 0,Y 488.095,Z 388.497,A -85,B 0,C 180,E1 -6679.34,E2 -6679.34} C_VEL
LIN {X 0,Y 488.089,Z 388.506,A -85,B 0,C 180,E1 -6680.62,E2 -6680.62} C_VEL
LIN {X 0,Y 488.095,Z 387.156,A -85,B 0,C 180,E1 -6681.985,E2 -6681.985} C_VEL
LIN {X 0,Y 488.214,Z 384.477,A -85,B 0,C 180,E1 -6683.32,E2 -6683.32} C_VEL
LIN {X 0,Y 488.352,Z 380.292,A -85,B 0,C 180,E1 -6684.667,E2 -6684.667} C_VEL
LIN {X 0,Y 488.481,Z 375.446,A -85,B 0,C 180,E1 -6685.799,E2 -6685.799} C_VEL
LIN {X 0,Y 488.629,Z 369.367,A -85,B 0,C 180,E1 -6686.906,E2 -6686.906} C_VEL
LIN {X 0,Y 488.843,Z 362.836,A -85,B 0,C 180,E1 -6687.855,E2 -6687.855} C_VEL
LIN {X 0,Y 489.086,Z 355.011,A -85,B 0,C 180,E1 -6688.771,E2 -6688.771} C_VEL
LIN {X 0,Y 489.327,Z 346.409,A -85,B 0,C 180,E1 -6689.584,E2 -6689.584} C_VEL
LIN {X 0,Y 489.633,Z 335.876,A -85,B 0,C 180,E1 -6690.36,E2 -6690.36} C_VEL
LIN {X 0,Y 489.841,Z 326.013,A -85,B 0,C 180,E1 -6690.919,E2 -6690.919} C_VEL
LIN {X 0,Y 490,Z 313.7,A -85,B 0,C 180,E1 -6691.417,E2 -6691.417} C_VEL
LIN {X 0,Y 490.111,Z 301.897,A -85,B 0,C 180,E1 -6691.711,E2 -6691.711} C_VEL
LIN {X 0,Y 490.594,Z 235.585,A -85,B 0,C 180,E1 -6692.76,E2 -6692.76} C_VEL
LIN {X 0,Y 489.004,Z 226.221,A -85,B 0,C 180,E1 -6692.978,E2 -6692.978} C_VEL
LIN {X 0,Y 488.966,Z 225.078,A -85,B 0,C 180,E1 -6693.105,E2 -6693.105} C_VEL
LIN {X 0,Y 489.23,Z 206.386,A -85,B 0,C 180,E1 -6696.728,E2 -6696.728} C_VEL
LIN {X 0,Y 489.247,Z 205.485,A -85,B 0,C 180,E1 -6696.902,E2 -6696.902} C_VEL
LIN {X 0,Y 488.661,Z 202.571,A -85,B 0,C 180,E1 -6697.498,E2 -6697.498} C_VEL
LIN {X 0,Y 483.156,Z 193.622,A -85,B 0,C 180,E1 -6699.487,E2 -6699.487} C_VEL
LIN {X 0,Y 482.483,Z 190.705,A -85,B 0,C 180,E1 -6700.097,E2 -6700.097} C_VEL
LIN {X 0,Y 482.052,Z 186.279,A -85,B 0,C 180,E1 -6701,E2 -6701} C_VEL
LIN {X 0,Y 481.741,Z 184.507,A -85,B 0,C 180,E1 -6701.438,E2 -6701.438} C_VEL
LIN {X 0,Y 481.653,Z 184.488,A -85,B 0,C 180,E1 -6704.457,E2 -6704.457} C_VEL
LIN {X 0,Y 481.646,Z 184.492,A -85,B 0,C 180,E1 -6707.839,E2 -6707.839} C_VEL
LIN {X 0,Y 481.659,Z 184.483,A -85,B 0,C 180,E1 -6710.654,E2 -6710.654} C_VEL
LIN {X 0,Y 481.629,Z 184.491,A -85,B 0,C 180,E1 -6713.375,E2 -6713.375} C_VEL
LIN {X 0,Y 481.708,Z 184.477,A -85,B 0,C 180,E1 -6716.33,E2 -6716.33} C_VEL
LIN {X 0,Y 481.649,Z 184.49,A -85,B 0,C 180,E1 -6719.417,E2 -6719.417} C_VEL
LIN {X 0,Y 481.7,Z 184.479,A -85,B 0,C 180,E1 -6722.168,E2 -6722.168} C_VEL
LIN {X 0,Y 481.716,Z 184.478,A -85,B 0,C 180,E1 -6724.969,E2 -6724.969} C_VEL
LIN {X 0,Y 481.648,Z 184.489,A -85,B 0,C 180,E1 -6727.704,E2 -6727.704} C_VEL
LIN {X 0,Y 481.703,Z 184.477,A -85,B 0,C 180,E1 -6730.393,E2 -6730.393} C_VEL
LIN {X 0,Y 481.687,Z 184.483,A -85,B 0,C 180,E1 -6733.033,E2 -6733.033} C_VEL
LIN {X 0,Y 481.692,Z 184.482,A -85,B 0,C 180,E1 -6735.638,E2 -6735.638} C_VEL
LIN {X 0,Y 481.749,Z 184.471,A -85,B 0,C 180,E1 -6738.215,E2 -6738.215} C_VEL
LIN {X 0,Y 481.761,Z 184.473,A -85,B 0,C 180,E1 -6741.611,E2 -6741.611} C_VEL
LIN {X 0,Y 481.817,Z 184.463,A -85,B 0,C 180,E1 -6744.139,E2 -6744.139} C_VEL
LIN {X 0,Y 481.926,Z 184.453,A -85,B 0,C 180,E1 -6747.492,E2 -6747.492} C_VEL
LIN {X 0,Y 481.903,Z 184.457,A -85,B 0,C 180,E1 -6750.835,E2 -6750.835} C_VEL
LIN {X 0,Y 481.926,Z 184.451,A -85,B 0,C 180,E1 -6752.507,E2 -6752.507} C_VEL
LIN {X 0,Y 481.805,Z 184.464,A -85,B 0,C 180,E1 -6755.86,E2 -6755.86} C_VEL
LIN {X 0,Y 481.759,Z 184.472,A -85,B 0,C 180,E1 -6758.388,E2 -6758.388} C_VEL
LIN {X 0,Y 481.747,Z 184.472,A -85,B 0,C 180,E1 -6761.784,E2 -6761.784} C_VEL
LIN {X 0,Y 481.738,Z 184.476,A -85,B 0,C 180,E1 -6765.224,E2 -6765.224} C_VEL
LIN {X 0,Y 481.708,Z 184.484,A -85,B 0,C 180,E1 -6768.721,E2 -6768.721} C_VEL
LIN {X 0,Y 481.642,Z 184.486,A -85,B 0,C 180,E1 -6771.394,E2 -6771.394} C_VEL
LIN {X 0,Y 481.672,Z 184.482,A -85,B 0,C 180,E1 -6774.112,E2 -6774.112} C_VEL
LIN {X 0,Y 481.746,Z 184.474,A -85,B 0,C 180,E1 -6777.14,E2 -6777.14} C_VEL
LIN {X 0,Y 481.673,Z 184.481,A -85,B 0,C 180,E1 -6779.74,E2 -6779.74} C_VEL
LIN {X 0,Y 481.667,Z 184.489,A -85,B 0,C 180,E1 -6782.673,E2 -6782.673} C_VEL
LIN {X 0,Y 481.637,Z 184.486,A -85,B 0,C 180,E1 -6785.708,E2 -6785.708} C_VEL
LIN {X 0,Y 481.707,Z 184.477,A -85,B 0,C 180,E1 -6789.353,E2 -6789.353} C_VEL
LIN {X 0,Y 481.666,Z 184.487,A -85,B 0,C 180,E1 -6792.157,E2 -6792.157} C_VEL
LIN {X 0,Y 481.652,Z 184.491,A -85,B 0,C 180,E1 -6794.457,E2 -6794.457} C_VEL
LIN {X 0,Y 481.641,Z 184.487,A -85,B 0,C 180,E1 -6797.839,E2 -6797.839} C_VEL
LIN {X 0,Y 481.706,Z 184.48,A -85,B 0,C 180,E1 -6800.646,E2 -6800.646} C_VEL
LIN {X 0,Y 481.635,Z 184.493,A -85,B 0,C 180,E1 -6804.291,E2 -6804.291} C_VEL
LIN {X 0,Y 481.665,Z 184.482,A -85,B 0,C 180,E1 -6807.326,E2 -6807.326} C_VEL
LIN {X 0,Y 481.68,Z 184.487,A -85,B 0,C 180,E1 -6810.259,E2 -6810.259} C_VEL
LIN {X 0,Y 481.737,Z 184.473,A -85,B 0,C 180,E1 -6813.112,E2 -6813.112} C_VEL
LIN {X 0,Y 481.669,Z 184.488,A -85,B 0,C 180,E1 -6815.887,E2 -6815.887} C_VEL
LIN {X 0,Y 481.693,Z 184.478,A -85,B 0,C 180,E1 -6819.027,E2 -6819.027} C_VEL
LIN {X 0,Y 481.699,Z 184.483,A -85,B 0,C 180,E1 -6822.159,E2 -6822.159} C_VEL
LIN {X 0,Y 481.733,Z 184.473,A -85,B 0,C 180,E1 -6824.776,E2 -6824.776} C_VEL
LIN {X 0,Y 481.744,Z 184.476,A -85,B 0,C 180,E1 -6828.215,E2 -6828.215} C_VEL
LIN {X 0,Y 481.755,Z 184.476,A -85,B 0,C 180,E1 -6831.612,E2 -6831.612} C_VEL
LIN {X 0,Y 481.807,Z 184.468,A -85,B 0,C 180,E1 -6834.14,E2 -6834.14} C_VEL
LIN {X 0,Y 481.919,Z 184.456,A -85,B 0,C 180,E1 -6837.493,E2 -6837.493} C_VEL
LIN {X 0,Y 481.897,Z 184.453,A -85,B 0,C 180,E1 -6840.836,E2 -6840.836} C_VEL
LIN {X 0,Y 481.919,Z 184.45,A -85,B 0,C 180,E1 -6842.508,E2 -6842.508} C_VEL
LIN {X 0,Y 481.799,Z 184.47,A -85,B 0,C 180,E1 -6845.861,E2 -6845.861} C_VEL
LIN {X 0,Y 481.753,Z 184.471,A -85,B 0,C 180,E1 -6848.389,E2 -6848.389} C_VEL
LIN {X 0,Y 481.743,Z 184.477,A -85,B 0,C 180,E1 -6851.786,E2 -6851.786} C_VEL
LIN {X 0,Y 481.735,Z 184.479,A -85,B 0,C 180,E1 -6855.225,E2 -6855.225} C_VEL
LIN {X 0,Y 481.705,Z 184.478,A -85,B 0,C 180,E1 -6858.722,E2 -6858.722} C_VEL
LIN {X 0,Y 481.639,Z 184.493,A -85,B 0,C 180,E1 -6861.395,E2 -6861.395} C_VEL
LIN {X 0,Y 481.663,Z 184.482,A -85,B 0,C 180,E1 -6864.114,E2 -6864.114} C_VEL
LIN {X 0,Y 481.739,Z 184.48,A -85,B 0,C 180,E1 -6867.14,E2 -6867.14} C_VEL
LIN {X 0,Y 481.672,Z 184.483,A -85,B 0,C 180,E1 -6869.742,E2 -6869.742} C_VEL
LIN {X 0,Y 481.664,Z 184.484,A -85,B 0,C 180,E1 -6872.675,E2 -6872.675} C_VEL
LIN {X 0,Y 481.63,Z 184.488,A -85,B 0,C 180,E1 -6875.711,E2 -6875.711} C_VEL
LIN {X 0,Y 481.665,Z 184.487,A -85,B 0,C 180,E1 -6878.86,E2 -6878.86} C_VEL
LIN {X 0,Y 481.648,Z 184.484,A -85,B 0,C 180,E1 -6881.914,E2 -6881.914} C_VEL
LIN {X 0,Y 481.656,Z 184.485,A -85,B 0,C 180,E1 -6884.458,E2 -6884.458} C_VEL
LIN {X 0,Y 481.639,Z 184.485,A -85,B 0,C 180,E1 -6887.84,E2 -6887.84} C_VEL
LIN {X 0,Y 481.657,Z 184.488,A -85,B 0,C 180,E1 -6890.655,E2 -6890.655} C_VEL
LIN {X 0,Y 481.619,Z 184.49,A -85,B 0,C 180,E1 -6893.378,E2 -6893.378} C_VEL
LIN {X 0,Y 481.692,Z 184.483,A -85,B 0,C 180,E1 -6896.33,E2 -6896.33} C_VEL
LIN {X 0,Y 481.647,Z 184.489,A -85,B 0,C 180,E1 -6899.419,E2 -6899.419} C_VEL
LIN {X 0,Y 481.672,Z 184.489,A -85,B 0,C 180,E1 -6902.565,E2 -6902.565} C_VEL
LIN {X 0,Y 481.74,Z 184.782,A -85,B 0,C 180,E1 -6902.964,E2 -6902.964} C_VEL
LIN {X 0,Y 485.007,Z 199.702,A -85,B 0,C 180,E1 -6905.152,E2 -6905.152} C_VEL
LIN {X 0,Y 483.999,Z 223.943,A -85,B 0,C 180,E1 -6908.33,E2 -6908.33} C_VEL
LIN {X 0,Y 483.012,Z 250.56,A -85,B 0,C 180,E1 -6911.771,E2 -6911.771} C_VEL
LIN {X 0,Y 482.526,Z 265.725,A -85,B 0,C 180,E1 -6913.696,E2 -6913.696} C_VEL
LIN {X 0,Y 482.988,Z 270.096,A -85,B 0,C 180,E1 -6913.817,E2 -6913.817} C_VEL
LIN {X 0,Y 484.328,Z 282.585,A -85,B 0,C 180,E1 -6914.051,E2 -6914.051} C_VEL
LIN {X 0,Y 483.678,Z 373.843,A -85,B 0,C 180,E1 -6915.458,E2 -6915.458} C_VEL
LIN {X 0,Y 483.402,Z 387.217,A -85,B 0,C 180,E1 -6915.826,E2 -6915.826} C_VEL
LIN {X 0,Y 483.034,Z 399.426,A -85,B 0,C 180,E1 -6916.325,E2 -6916.325} C_VEL
LIN {X 0,Y 482.634,Z 410.906,A -85,B 0,C 180,E1 -6916.956,E2 -6916.956} C_VEL
LIN {X 0,Y 482.325,Z 422.218,A -85,B 0,C 180,E1 -6917.764,E2 -6917.764} C_VEL
LIN {X 0,Y 481.792,Z 433.265,A -85,B 0,C 180,E1 -6918.75,E2 -6918.75} C_VEL
LIN {X 0,Y 481.538,Z 441.904,A -85,B 0,C 180,E1 -6919.702,E2 -6919.702} C_VEL
LIN {X 0,Y 481.316,Z 449.845,A -85,B 0,C 180,E1 -6920.758,E2 -6920.758} C_VEL
LIN {X 0,Y 481.145,Z 457.576,A -85,B 0,C 180,E1 -6922.024,E2 -6922.024} C_VEL
LIN {X 0,Y 481.013,Z 463.774,A -85,B 0,C 180,E1 -6923.288,E2 -6923.288} C_VEL
LIN {X 0,Y 480.99,Z 468.674,A -85,B 0,C 180,E1 -6924.551,E2 -6924.551} C_VEL
LIN {X 0,Y 480.988,Z 472.415,A -85,B 0,C 180,E1 -6925.811,E2 -6925.811} C_VEL
LIN {X 0,Y 481.033,Z 474.341,A -85,B 0,C 180,E1 -6926.65,E2 -6926.65} C_VEL
LIN {X 0,Y 480.955,Z 475.784,A -85,B 0,C 180,E1 -6927.488,E2 -6927.488} C_VEL
LIN {X 0,Y 480.87,Z 477.403,A -85,B 0,C 180,E1 -6929.163,E2 -6929.163} C_VEL
LIN {X 0,Y 480.885,Z 477.611,A -85,B 0,C 180,E1 -6930.001,E2 -6930.001} C_VEL
LIN {X 0,Y 480.874,Z 477.364,A -85,B 0,C 180,E1 -6930.838,E2 -6930.838} C_VEL
LIN {X 0,Y 480.957,Z 475.658,A -85,B 0,C 180,E1 -6932.513,E2 -6932.513} C_VEL
LIN {X 0,Y 481.047,Z 474.181,A -85,B 0,C 180,E1 -6933.351,E2 -6933.351} C_VEL
LIN {X 0,Y 480.918,Z 471.075,A -85,B 0,C 180,E1 -6934.611,E2 -6934.611} C_VEL
LIN {X 0,Y 481,Z 466.898,A -85,B 0,C 180,E1 -6935.871,E2 -6935.871} C_VEL
LIN {X 0,Y 481.099,Z 460.47,A -85,B 0,C 180,E1 -6937.344,E2 -6937.344} C_VEL
LIN {X 0,Y 481.183,Z 453.461,A -85,B 0,C 180,E1 -6938.611,E2 -6938.611} C_VEL
LIN {X 0,Y 481.355,Z 446.308,A -85,B 0,C 180,E1 -6939.667,E2 -6939.667} C_VEL
LIN {X 0,Y 481.66,Z 437.69,A -85,B 0,C 180,E1 -6940.722,E2 -6940.722} C_VEL
LIN {X 0,Y 482.035,Z 427.015,A -85,B 0,C 180,E1 -6941.778,E2 -6941.778} C_VEL
LIN {X 0,Y 482.345,Z 416.426,A -85,B 0,C 180,E1 -6942.625,E2 -6942.625} C_VEL
LIN {X 0,Y 482.765,Z 404.797,A -85,B 0,C 180,E1 -6943.363,E2 -6943.363} C_VEL
LIN {X 0,Y 483.177,Z 392.707,A -85,B 0,C 180,E1 -6943.941,E2 -6943.941} C_VEL
LIN {X 0,Y 483.558,Z 379.598,A -85,B 0,C 180,E1 -6944.386,E2 -6944.386} C_VEL
LIN {X 0,Y 483.761,Z 367.114,A -85,B 0,C 180,E1 -6944.648,E2 -6944.648} C_VEL
LIN {X 0,Y 484.236,Z 280.809,A -85,B 0,C 180,E1 -6945.992,E2 -6945.992} C_VEL
LIN {X 0,Y 482.482,Z 264.96,A -85,B 0,C 180,E1 -6946.331,E2 -6946.331} C_VEL
LIN {X 0,Y 483.176,Z 240.407,A -85,B 0,C 180,E1 -6949.367,E2 -6949.367} C_VEL
LIN {X 0,Y 483.955,Z 214.442,A -85,B 0,C 180,E1 -6952.634,E2 -6952.634} C_VEL
LIN {X 0,Y 484.531,Z 198.579,A -85,B 0,C 180,E1 -6954.646,E2 -6954.646} C_VEL
LIN {X 0,Y 482.835,Z 189.624,A -85,B 0,C 180,E1 -6955.892,E2 -6955.892} C_VEL
LIN {X 0,Y 481.693,Z 184.602,A -85,B 0,C 180,E1 -6956.657,E2 -6956.657} C_VEL
LIN {X 0,Y 481.67,Z 184.489,A -85,B 0,C 180,E1 -6959.742,E2 -6959.742} C_VEL
LIN {X 0,Y 481.673,Z 184.487,A -85,B 0,C 180,E1 -6962.674,E2 -6962.674} C_VEL
LIN {X 0,Y 481.634,Z 184.491,A -85,B 0,C 180,E1 -6965.71,E2 -6965.71} C_VEL
LIN {X 0,Y 481.668,Z 184.488,A -85,B 0,C 180,E1 -6968.86,E2 -6968.86} C_VEL
LIN {X 0,Y 481.632,Z 184.489,A -85,B 0,C 180,E1 -6972.163,E2 -6972.163} C_VEL
LIN {X 0,Y 481.656,Z 184.486,A -85,B 0,C 180,E1 -6975.542,E2 -6975.542} C_VEL
LIN {X 0,Y 481.65,Z 184.492,A -85,B 0,C 180,E1 -6978.957,E2 -6978.957} C_VEL
LIN {X 0,Y 481.656,Z 184.484,A -85,B 0,C 180,E1 -6981.993,E2 -6981.993} C_VEL
LIN {X 0,Y 481.687,Z 184.483,A -85,B 0,C 180,E1 -6985.317,E2 -6985.317} C_VEL
LIN {X 0,Y 481.646,Z 184.488,A -85,B 0,C 180,E1 -6988.311,E2 -6988.311} C_VEL
LIN {X 0,Y 481.699,Z 184.482,A -85,B 0,C 180,E1 -6991.218,E2 -6991.218} C_VEL
LIN {X 0,Y 481.691,Z 184.482,A -85,B 0,C 180,E1 -6994.042,E2 -6994.042} C_VEL
LIN {X 0,Y 481.676,Z 184.486,A -85,B 0,C 180,E1 -6996.812,E2 -6996.812} C_VEL
LIN {X 0,Y 481.697,Z 184.48,A -85,B 0,C 180,E1 -6999.502,E2 -6999.502} C_VEL
LIN {X 0,Y 481.69,Z 184.484,A -85,B 0,C 180,E1 -7002.157,E2 -7002.157} C_VEL
LIN {X 0,Y 481.744,Z 184.479,A -85,B 0,C 180,E1 -7004.775,E2 -7004.775} C_VEL
LIN {X 0,Y 481.752,Z 184.478,A -85,B 0,C 180,E1 -7008.215,E2 -7008.215} C_VEL
LIN {X 0,Y 481.742,Z 184.476,A -85,B 0,C 180,E1 -7011.611,E2 -7011.611} C_VEL
LIN {X 0,Y 481.797,Z 184.473,A -85,B 0,C 180,E1 -7014.139,E2 -7014.139} C_VEL
LIN {X 0,Y 481.927,Z 184.455,A -85,B 0,C 180,E1 -7017.492,E2 -7017.492} C_VEL
LIN {X 0,Y 481.943,Z 184.673,A -85,B 0,C 180,E1 -7019.53,E2 -7019.53} C_VEL
LIN {X 0,Y 482.264,Z 189.786,A -85,B 0,C 180,E1 -7020.417,E2 -7020.417} C_VEL
LIN {X 0,Y 482.169,Z 205.875,A -85,B 0,C 180,E1 -7023.133,E2 -7023.133} C_VEL
LIN {X 0,Y 482.146,Z 221.491,A -85,B 0,C 180,E1 -7025.856,E2 -7025.856} C_VEL
LIN {X 0,Y 482.165,Z 226.715,A -85,B 0,C 180,E1 -7026.731,E2 -7026.731} C_VEL
LIN {X 0,Y 484.041,Z 237.633,A -85,B 0,C 180,E1 -7027.016,E2 -7027.016} C_VEL
LIN {X 0,Y 483.301,Z 307.943,A -85,B 0,C 180,E1 -7028.236,E2 -7028.236} C_VEL
LIN {X 0,Y 483.187,Z 319.489,A -85,B 0,C 180,E1 -7028.6,E2 -7028.6} C_VEL
LIN {X 0,Y 482.978,Z 331.146,A -85,B 0,C 180,E1 -7029.152,E2 -7029.152} C_VEL
LIN {X 0,Y 482.697,Z 341.903,A -85,B 0,C 180,E1 -7029.85,E2 -7029.85} C_VEL
LIN {X 0,Y 482.384,Z 351.993,A -85,B 0,C 180,E1 -7030.705,E2 -7030.705} C_VEL
LIN {X 0,Y 482.132,Z 359.964,A -85,B 0,C 180,E1 -7031.562,E2 -7031.562} C_VEL
LIN {X 0,Y 481.834,Z 367.977,A -85,B 0,C 180,E1 -7032.637,E2 -7032.637} C_VEL
LIN {X 0,Y 481.633,Z 374.293,A -85,B 0,C 180,E1 -7033.716,E2 -7033.716} C_VEL
LIN {X 0,Y 481.447,Z 379.321,A -85,B 0,C 180,E1 -7034.8,E2 -7034.8} C_VEL
LIN {X 0,Y 481.273,Z 383.847,A -85,B 0,C 180,E1 -7036.108,E2 -7036.108} C_VEL
LIN {X 0,Y 481.176,Z 386.085,A -85,B 0,C 180,E1 -7036.984,E2 -7036.984} C_VEL
LIN {X 0,Y 481.054,Z 388.265,A -85,B 0,C 180,E1 -7038.264,E2 -7038.264} C_VEL
LIN {X 0,Y 481.045,Z 389.265,A -85,B 0,C 180,E1 -7039.635,E2 -7039.635} C_VEL
LIN {X 0,Y 481.016,Z 389.074,A -85,B 0,C 180,E1 -7040.758,E2 -7040.758} C_VEL
LIN {X 0,Y 481.019,Z 388.531,A -85,B 0,C 180,E1 -7041.424,E2 -7041.424} C_VEL
LIN {X 0,Y 481.053,Z 387.297,A -85,B 0,C 180,E1 -7042.324,E2 -7042.324} C_VEL
LIN {X 0,Y 481.208,Z 384.268,A -85,B 0,C 180,E1 -7043.68,E2 -7043.68} C_VEL
LIN {X 0,Y 481.308,Z 379.655,A -85,B 0,C 180,E1 -7045.052,E2 -7045.052} C_VEL
LIN {X 0,Y 481.48,Z 374.447,A -85,B 0,C 180,E1 -7046.202,E2 -7046.202} C_VEL
LIN {X 0,Y 481.706,Z 367.223,A -85,B 0,C 180,E1 -7047.425,E2 -7047.425} C_VEL
LIN {X 0,Y 481.978,Z 358.865,A -85,B 0,C 180,E1 -7048.525,E2 -7048.525} C_VEL
LIN {X 0,Y 482.269,Z 349.628,A -85,B 0,C 180,E1 -7049.48,E2 -7049.48} C_VEL
LIN {X 0,Y 482.573,Z 339.7,A -85,B 0,C 180,E1 -7050.282,E2 -7050.282} C_VEL
LIN {X 0,Y 482.817,Z 328.575,A -85,B 0,C 180,E1 -7050.966,E2 -7050.966} C_VEL
LIN {X 0,Y 483.048,Z 317.21,A -85,B 0,C 180,E1 -7051.472,E2 -7051.472} C_VEL
LIN {X 0,Y 483.162,Z 304.584,A -85,B 0,C 180,E1 -7051.837,E2 -7051.837} C_VEL
LIN {X 0,Y 483.626,Z 235.755,A -85,B 0,C 180,E1 -7052.958,E2 -7052.958} C_VEL
LIN {X 0,Y 481.987,Z 226.138,A -85,B 0,C 180,E1 -7053.195,E2 -7053.195} C_VEL
LIN {X 0,Y 481.987,Z 220.794,A -85,B 0,C 180,E1 -7054.175,E2 -7054.175} C_VEL
LIN {X 0,Y 482.299,Z 205.284,A -85,B 0,C 180,E1 -7057.208,E2 -7057.208} C_VEL
LIN {X 0,Y 482.483,Z 190.705,A -85,B 0,C 180,E1 -7060.097,E2 -7060.097} C_VEL
LIN {X 0,Y 481.706,Z 188.844,A -85,B 0,C 180,E1 -7060.509,E2 -7060.509} C_VEL
LIN {X 0,Y 478.554,Z 186.677,A -85,B 0,C 180,E1 -7061.183,E2 -7061.183} C_VEL
LIN {X 0,Y 475.396,Z 185.56,A -85,B 0,C 180,E1 -7061.9,E2 -7061.9} C_VEL
LIN {X 0,Y 474.624,Z 185.363,A -85,B 0,C 180,E1 -7062.377,E2 -7062.377} C_VEL
LIN {X 0,Y 474.615,Z 185.365,A -85,B 0,C 180,E1 -7065.297,E2 -7065.297} C_VEL
LIN {X 0,Y 474.619,Z 185.363,A -85,B 0,C 180,E1 -7068.214,E2 -7068.214} C_VEL
LIN {X 0,Y 474.61,Z 185.367,A -85,B 0,C 180,E1 -7071.542,E2 -7071.542} C_VEL
LIN {X 0,Y 474.627,Z 185.359,A -85,B 0,C 180,E1 -7074.726,E2 -7074.726} C_VEL
LIN {X 0,Y 474.634,Z 185.363,A -85,B 0,C 180,E1 -7077.787,E2 -7077.787} C_VEL
LIN {X 0,Y 474.622,Z 185.36,A -85,B 0,C 180,E1 -7080.884,E2 -7080.884} C_VEL
LIN {X 0,Y 474.666,Z 185.36,A -85,B 0,C 180,E1 -7083.628,E2 -7083.628} C_VEL
LIN {X 0,Y 474.634,Z 185.358,A -85,B 0,C 180,E1 -7086.641,E2 -7086.641} C_VEL
LIN {X 0,Y 474.653,Z 185.356,A -85,B 0,C 180,E1 -7090.089,E2 -7090.089} C_VEL
LIN {X 0,Y 474.646,Z 185.358,A -85,B 0,C 180,E1 -7092.774,E2 -7092.774} C_VEL
LIN {X 0,Y 474.65,Z 185.363,A -85,B 0,C 180,E1 -7095.421,E2 -7095.421} C_VEL
LIN {X 0,Y 474.702,Z 185.35,A -85,B 0,C 180,E1 -7098.037,E2 -7098.037} C_VEL
LIN {X 0,Y 474.726,Z 185.351,A -85,B 0,C 180,E1 -7101.486,E2 -7101.486} C_VEL
LIN {X 0,Y 474.779,Z 185.34,A -85,B 0,C 180,E1 -7104.052,E2 -7104.052} C_VEL
LIN {X 0,Y 474.892,Z 185.329,A -85,B 0,C 180,E1 -7107.455,E2 -7107.455} C_VEL
LIN {X 0,Y 474.91,Z 185.323,A -85,B 0,C 180,E1 -7109.999,E2 -7109.999} C_VEL
LIN {X 0,Y 474.892,Z 185.328,A -85,B 0,C 180,E1 -7112.544,E2 -7112.544} C_VEL
LIN {X 0,Y 474.768,Z 185.341,A -85,B 0,C 180,E1 -7115.947,E2 -7115.947} C_VEL
LIN {X 0,Y 474.725,Z 185.349,A -85,B 0,C 180,E1 -7118.513,E2 -7118.513} C_VEL
LIN {X 0,Y 474.7,Z 185.349,A -85,B 0,C 180,E1 -7121.962,E2 -7121.962} C_VEL
LIN {X 0,Y 474.696,Z 185.351,A -85,B 0,C 180,E1 -7125.455,E2 -7125.455} C_VEL
LIN {X 0,Y 474.661,Z 185.36,A -85,B 0,C 180,E1 -7129.01,E2 -7129.01} C_VEL
LIN {X 0,Y 474.585,Z 185.364,A -85,B 0,C 180,E1 -7131.728,E2 -7131.728} C_VEL
LIN {X 0,Y 474.654,Z 185.361,A -85,B 0,C 180,E1 -7134.492,E2 -7134.492} C_VEL
LIN {X 0,Y 474.693,Z 185.351,A -85,B 0,C 180,E1 -7137.338,E2 -7137.338} C_VEL
LIN {X 0,Y 474.599,Z 185.368,A -85,B 0,C 180,E1 -7140.81,E2 -7140.81} C_VEL
LIN {X 0,Y 474.632,Z 185.36,A -85,B 0,C 180,E1 -7143.984,E2 -7143.984} C_VEL
LIN {X 0,Y 474.569,Z 185.369,A -85,B 0,C 180,E1 -7146.9,E2 -7146.9} C_VEL
LIN {X 0,Y 474.643,Z 185.357,A -85,B 0,C 180,E1 -7149.651,E2 -7149.651} C_VEL
LIN {X 0,Y 474.644,Z 185.359,A -85,B 0,C 180,E1 -7152.93,E2 -7152.93} C_VEL
LIN {X 0,Y 474.601,Z 185.364,A -85,B 0,C 180,E1 -7155.895,E2 -7155.895} C_VEL
LIN {X 0,Y 474.633,Z 185.359,A -85,B 0,C 180,E1 -7159.039,E2 -7159.039} C_VEL
LIN {X 0,Y 474.608,Z 185.363,A -85,B 0,C 180,E1 -7161.703,E2 -7161.703} C_VEL
LIN {X 0,Y 474.622,Z 185.361,A -85,B 0,C 180,E1 -7164.726,E2 -7164.726} C_VEL
LIN {X 0,Y 474.629,Z 185.362,A -85,B 0,C 180,E1 -7167.788,E2 -7167.788} C_VEL
LIN {X 0,Y 474.623,Z 185.36,A -85,B 0,C 180,E1 -7170.883,E2 -7170.883} C_VEL
LIN {X 0,Y 474.651,Z 185.358,A -85,B 0,C 180,E1 -7173.628,E2 -7173.628} C_VEL
LIN {X 0,Y 474.627,Z 185.36,A -85,B 0,C 180,E1 -7176.641,E2 -7176.641} C_VEL
LIN {X 0,Y 474.648,Z 185.363,A -85,B 0,C 180,E1 -7180.09,E2 -7180.09} C_VEL
LIN {X 0,Y 474.642,Z 185.357,A -85,B 0,C 180,E1 -7182.775,E2 -7182.775} C_VEL
LIN {X 0,Y 474.639,Z 185.359,A -85,B 0,C 180,E1 -7185.421,E2 -7185.421} C_VEL
LIN {X 0,Y 474.697,Z 185.356,A -85,B 0,C 180,E1 -7188.038,E2 -7188.038} C_VEL
LIN {X 0,Y 474.72,Z 185.351,A -85,B 0,C 180,E1 -7191.487,E2 -7191.487} C_VEL
LIN {X 0,Y 474.77,Z 185.345,A -85,B 0,C 180,E1 -7194.053,E2 -7194.053} C_VEL
LIN {X 0,Y 474.885,Z 185.331,A -85,B 0,C 180,E1 -7197.456,E2 -7197.456} C_VEL
LIN {X 0,Y 474.902,Z 185.328,A -85,B 0,C 180,E1 -7200,E2 -7200} C_VEL
LIN {X 0,Y 474.885,Z 185.327,A -85,B 0,C 180,E1 -7202.545,E2 -7202.545} C_VEL
LIN {X 0,Y 474.762,Z 185.345,A -85,B 0,C 180,E1 -7205.948,E2 -7205.948} C_VEL
LIN {X 0,Y 474.719,Z 185.347,A -85,B 0,C 180,E1 -7208.514,E2 -7208.514} C_VEL
LIN {X 0,Y 474.696,Z 185.352,A -85,B 0,C 180,E1 -7211.963,E2 -7211.963} C_VEL
LIN {X 0,Y 474.692,Z 185.359,A -85,B 0,C 180,E1 -7215.456,E2 -7215.456} C_VEL
LIN {X 0,Y 474.657,Z 185.358,A -85,B 0,C 180,E1 -7219.011,E2 -7219.011} C_VEL
LIN {X 0,Y 474.581,Z 185.368,A -85,B 0,C 180,E1 -7221.73,E2 -7221.73} C_VEL
LIN {X 0,Y 474.647,Z 185.356,A -85,B 0,C 180,E1 -7224.494,E2 -7224.494} C_VEL
LIN {X 0,Y 474.674,Z 185.36,A -85,B 0,C 180,E1 -7227.335,E2 -7227.335} C_VEL
LIN {X 0,Y 474.598,Z 185.366,A -85,B 0,C 180,E1 -7230.811,E2 -7230.811} C_VEL
LIN {X 0,Y 474.619,Z 185.367,A -85,B 0,C 180,E1 -7233.222,E2 -7233.222} C_VEL
LIN {X 0,Y 474.583,Z 185.364,A -85,B 0,C 180,E1 -7236.324,E2 -7236.324} C_VEL
LIN {X 0,Y 474.613,Z 185.362,A -85,B 0,C 180,E1 -7239.647,E2 -7239.647} C_VEL
LIN {X 0,Y 474.62,Z 185.36,A -85,B 0,C 180,E1 -7242.238,E2 -7242.238} C_VEL
LIN {X 0,Y 474.617,Z 185.364,A -85,B 0,C 180,E1 -7245.298,E2 -7245.298} C_VEL
LIN {X 0,Y 474.61,Z 185.361,A -85,B 0,C 180,E1 -7248.215,E2 -7248.215} C_VEL
LIN {X 0,Y 474.607,Z 185.362,A -85,B 0,C 180,E1 -7251.544,E2 -7251.544} C_VEL
LIN {X 0,Y 474.62,Z 185.367,A -85,B 0,C 180,E1 -7254.726,E2 -7254.726} C_VEL
LIN {X 0,Y 474.634,Z 185.361,A -85,B 0,C 180,E1 -7257.789,E2 -7257.789} C_VEL
LIN {X 0,Y 474.606,Z 185.368,A -85,B 0,C 180,E1 -7260.889,E2 -7260.889} C_VEL
LIN {X 0,Y 474.664,Z 185.55,A -85,B 0,C 180,E1 -7262.699,E2 -7262.699} C_VEL
LIN {X 0,Y 478.082,Z 200.884,A -85,B 0,C 180,E1 -7265,E2 -7265} C_VEL
LIN {X 0,Y 477.179,Z 222.802,A -85,B 0,C 180,E1 -7267.92,E2 -7267.92} C_VEL
LIN {X 0,Y 476.061,Z 250.057,A -85,B 0,C 180,E1 -7271.495,E2 -7271.495} C_VEL
LIN {X 0,Y 475.538,Z 265.538,A -85,B 0,C 180,E1 -7273.494,E2 -7273.494} C_VEL
LIN {X 0,Y 477.44,Z 282.568,A -85,B 0,C 180,E1 -7273.849,E2 -7273.849} C_VEL
LIN {X 0,Y 476.738,Z 374.186,A -85,B 0,C 180,E1 -7275.296,E2 -7275.296} C_VEL
LIN {X 0,Y 476.414,Z 388.028,A -85,B 0,C 180,E1 -7275.695,E2 -7275.695} C_VEL
LIN {X 0,Y 476.01,Z 400.411,A -85,B 0,C 180,E1 -7276.228,E2 -7276.228} C_VEL
LIN {X 0,Y 475.524,Z 413.075,A -85,B 0,C 180,E1 -7276.975,E2 -7276.975} C_VEL
LIN {X 0,Y 475.236,Z 423.391,A -85,B 0,C 180,E1 -7277.754,E2 -7277.754} C_VEL
LIN {X 0,Y 474.715,Z 433.459,A -85,B 0,C 180,E1 -7278.688,E2 -7278.688} C_VEL
LIN {X 0,Y 474.423,Z 442.785,A -85,B 0,C 180,E1 -7279.761,E2 -7279.761} C_VEL
LIN {X 0,Y 474.167,Z 451.841,A -85,B 0,C 180,E1 -7281.047,E2 -7281.047} C_VEL
LIN {X 0,Y 474.001,Z 459.1,A -85,B 0,C 180,E1 -7282.332,E2 -7282.332} C_VEL
LIN {X 0,Y 473.855,Z 465.692,A -85,B 0,C 180,E1 -7283.832,E2 -7283.832} C_VEL
LIN {X 0,Y 473.848,Z 469.369,A -85,B 0,C 180,E1 -7284.895,E2 -7284.895} C_VEL
LIN {X 0,Y 473.884,Z 471.744,A -85,B 0,C 180,E1 -7285.748,E2 -7285.748} C_VEL
LIN {X 0,Y 473.952,Z 473.678,A -85,B 0,C 180,E1 -7286.6,E2 -7286.6} C_VEL
LIN {X 0,Y 473.897,Z 475.132,A -85,B 0,C 180,E1 -7287.451,E2 -7287.451} C_VEL
LIN {X 0,Y 473.799,Z 476.753,A -85,B 0,C 180,E1 -7289.151,E2 -7289.151} C_VEL
LIN {X 0,Y 473.815,Z 476.961,A -85,B 0,C 180,E1 -7290.001,E2 -7290.001} C_VEL
LIN {X 0,Y 473.802,Z 476.713,A -85,B 0,C 180,E1 -7290.85,E2 -7290.85} C_VEL
LIN {X 0,Y 473.9,Z 475.003,A -85,B 0,C 180,E1 -7292.551,E2 -7292.551} C_VEL
LIN {X 0,Y 473.966,Z 473.518,A -85,B 0,C 180,E1 -7293.401,E2 -7293.401} C_VEL
LIN {X 0,Y 473.829,Z 470.403,A -85,B 0,C 180,E1 -7294.68,E2 -7294.68} C_VEL
LIN {X 0,Y 473.892,Z 466.212,A -85,B 0,C 180,E1 -7295.959,E2 -7295.959} C_VEL
LIN {X 0,Y 474.001,Z 459.764,A -85,B 0,C 180,E1 -7297.455,E2 -7297.455} C_VEL
LIN {X 0,Y 474.107,Z 452.734,A -85,B 0,C 180,E1 -7298.74,E2 -7298.74} C_VEL
LIN {X 0,Y 474.284,Z 445.566,A -85,B 0,C 180,E1 -7299.812,E2 -7299.812} C_VEL
LIN {X 0,Y 474.633,Z 436.928,A -85,B 0,C 180,E1 -7300.883,E2 -7300.883} C_VEL
LIN {X 0,Y 474.985,Z 427.422,A -85,B 0,C 180,E1 -7301.847,E2 -7301.847} C_VEL
LIN {X 0,Y 475.366,Z 415.609,A -85,B 0,C 180,E1 -7302.813,E2 -7302.813} C_VEL
LIN {X 0,Y 475.8,Z 403.902,A -85,B 0,C 180,E1 -7303.562,E2 -7303.562} C_VEL
LIN {X 0,Y 476.282,Z 391.716,A -85,B 0,C 180,E1 -7304.147,E2 -7304.147} C_VEL
LIN {X 0,Y 476.693,Z 378.47,A -85,B 0,C 180,E1 -7304.597,E2 -7304.597} C_VEL
LIN {X 0,Y 476.869,Z 365.537,A -85,B 0,C 180,E1 -7304.865,E2 -7304.865} C_VEL
LIN {X 0,Y 477.402,Z 281.643,A -85,B 0,C 180,E1 -7306.201,E2 -7306.201} C_VEL
LIN {X 0,Y 475.535,Z 264.748,A -85,B 0,C 180,E1 -7306.558,E2 -7306.558} C_VEL
LIN {X 0,Y 476.197,Z 241.903,A -85,B 0,C 180,E1 -7309.421,E2 -7309.421} C_VEL
LIN {X 0,Y 477.01,Z 217.533,A -85,B 0,C 180,E1 -7312.524,E2 -7312.524} C_VEL
LIN {X 0,Y 477.684,Z 199.977,A -85,B 0,C 180,E1 -7314.791,E2 -7314.791} C_VEL
LIN {X 0,Y 475.562,Z 189.268,A -85,B 0,C 180,E1 -7316.318,E2 -7316.318} C_VEL
LIN {X 0,Y 474.664,Z 185.501,A -85,B 0,C 180,E1 -7316.906,E2 -7316.906} C_VEL
LIN {X 0,Y 474.6,Z 185.367,A -85,B 0,C 180,E1 -7320.231,E2 -7320.231} C_VEL
LIN {X 0,Y 474.628,Z 185.367,A -85,B 0,C 180,E1 -7323.222,E2 -7323.222} C_VEL
LIN {X 0,Y 474.587,Z 185.367,A -85,B 0,C 180,E1 -7326.324,E2 -7326.324} C_VEL
LIN {X 0,Y 474.624,Z 185.364,A -85,B 0,C 180,E1 -7329.548,E2 -7329.548} C_VEL
LIN {X 0,Y 474.591,Z 185.366,A -85,B 0,C 180,E1 -7332.232,E2 -7332.232} C_VEL
LIN {X 0,Y 474.619,Z 185.365,A -85,B 0,C 180,E1 -7335.298,E2 -7335.298} C_VEL
LIN {X 0,Y 474.616,Z 185.361,A -85,B 0,C 180,E1 -7338.214,E2 -7338.214} C_VEL
LIN {X 0,Y 474.613,Z 185.362,A -85,B 0,C 180,E1 -7341.542,E2 -7341.542} C_VEL
LIN {X 0,Y 474.625,Z 185.365,A -85,B 0,C 180,E1 -7344.725,E2 -7344.725} C_VEL
LIN {X 0,Y 474.637,Z 185.359,A -85,B 0,C 180,E1 -7347.787,E2 -7347.787} C_VEL
LIN {X 0,Y 474.624,Z 185.365,A -85,B 0,C 180,E1 -7350.885,E2 -7350.885} C_VEL
LIN {X 0,Y 474.655,Z 185.357,A -85,B 0,C 180,E1 -7353.628,E2 -7353.628} C_VEL
LIN {X 0,Y 474.636,Z 185.364,A -85,B 0,C 180,E1 -7356.641,E2 -7356.641} C_VEL
LIN {X 0,Y 474.655,Z 185.359,A -85,B 0,C 180,E1 -7360.089,E2 -7360.089} C_VEL
LIN {X 0,Y 474.637,Z 185.364,A -85,B 0,C 180,E1 -7362.774,E2 -7362.774} C_VEL
LIN {X 0,Y 474.647,Z 185.359,A -85,B 0,C 180,E1 -7365.421,E2 -7365.421} C_VEL
LIN {X 0,Y 474.706,Z 185.354,A -85,B 0,C 180,E1 -7368.037,E2 -7368.037} C_VEL
LIN {X 0,Y 474.713,Z 185.351,A -85,B 0,C 180,E1 -7371.486,E2 -7371.486} C_VEL
LIN {X 0,Y 474.745,Z 185.35,A -85,B 0,C 180,E1 -7374.904,E2 -7374.904} C_VEL
LIN {X 0,Y 474.893,Z 185.332,A -85,B 0,C 180,E1 -7377.455,E2 -7377.455} C_VEL
LIN {X 0,Y 474.888,Z 185.478,A -85,B 0,C 180,E1 -7379.311,E2 -7379.311} C_VEL
LIN {X 0,Y 475.383,Z 189.329,A -85,B 0,C 180,E1 -7380,E2 -7380} C_VEL
LIN {X 0,Y 475.238,Z 206.719,A -85,B 0,C 180,E1 -7382.967,E2 -7382.967} C_VEL
LIN {X 0,Y 475.199,Z 222.481,A -85,B 0,C 180,E1 -7385.729,E2 -7385.729} C_VEL
LIN {X 0,Y 475.226,Z 226.906,A -85,B 0,C 180,E1 -7386.474,E2 -7386.474} C_VEL
LIN {X 0,Y 477.136,Z 237.294,A -85,B 0,C 180,E1 -7386.767,E2 -7386.767} C_VEL
LIN {X 0,Y 476.434,Z 308.978,A -85,B 0,C 180,E1 -7388.056,E2 -7388.056} C_VEL
LIN {X 0,Y 476.303,Z 320.385,A -85,B 0,C 180,E1 -7388.427,E2 -7388.427} C_VEL
LIN {X 0,Y 476.049,Z 332.623,A -85,B 0,C 180,E1 -7389.024,E2 -7389.024} C_VEL
LIN {X 0,Y 475.719,Z 343.805,A -85,B 0,C 180,E1 -7389.781,E2 -7389.781} C_VEL
LIN {X 0,Y 475.396,Z 353.585,A -85,B 0,C 180,E1 -7390.649,E2 -7390.649} C_VEL
LIN {X 0,Y 475.12,Z 361.411,A -85,B 0,C 180,E1 -7391.519,E2 -7391.519} C_VEL
LIN {X 0,Y 474.834,Z 368.695,A -85,B 0,C 180,E1 -7392.524,E2 -7392.524} C_VEL
LIN {X 0,Y 474.592,Z 375.458,A -85,B 0,C 180,E1 -7393.705,E2 -7393.705} C_VEL
LIN {X 0,Y 474.333,Z 381.204,A -85,B 0,C 180,E1 -7395.028,E2 -7395.028} C_VEL
LIN {X 0,Y 474.198,Z 385.394,A -85,B 0,C 180,E1 -7396.355,E2 -7396.355} C_VEL
LIN {X 0,Y 474.08,Z 387.409,A -85,B 0,C 180,E1 -7397.246,E2 -7397.246} C_VEL
LIN {X 0,Y 473.985,Z 389.126,A -85,B 0,C 180,E1 -7398.385,E2 -7398.385} C_VEL
LIN {X 0,Y 473.968,Z 389.68,A -85,B 0,C 180,E1 -7399.039,E2 -7399.039} C_VEL
LIN {X 0,Y 473.962,Z 389.962,A -85,B 0,C 180,E1 -7399.94,E2 -7399.94} C_VEL
LIN {X 0,Y 473.945,Z 389.635,A -85,B 0,C 180,E1 -7400.899,E2 -7400.899} C_VEL
LIN {X 0,Y 473.983,Z 388.816,A -85,B 0,C 180,E1 -7401.758,E2 -7401.758} C_VEL
LIN {X 0,Y 474.098,Z 386.21,A -85,B 0,C 180,E1 -7403.208,E2 -7403.208} C_VEL
LIN {X 0,Y 474.223,Z 382.465,A -85,B 0,C 180,E1 -7404.516,E2 -7404.516} C_VEL
LIN {X 0,Y 474.366,Z 377.913,A -85,B 0,C 180,E1 -7405.68,E2 -7405.68} C_VEL
LIN {X 0,Y 474.535,Z 371.96,A -85,B 0,C 180,E1 -7406.853,E2 -7406.853} C_VEL
LIN {X 0,Y 474.813,Z 364.459,A -85,B 0,C 180,E1 -7408.007,E2 -7408.007} C_VEL
LIN {X 0,Y 475.104,Z 356.471,A -85,B 0,C 180,E1 -7408.976,E2 -7408.976} C_VEL
LIN {X 0,Y 475.378,Z 346.864,A -85,B 0,C 180,E1 -7409.906,E2 -7409.906} C_VEL
LIN {X 0,Y 475.717,Z 337.055,A -85,B 0,C 180,E1 -7410.642,E2 -7410.642} C_VEL
LIN {X 0,Y 475.947,Z 326.725,A -85,B 0,C 180,E1 -7411.242,E2 -7411.242} C_VEL
LIN {X 0,Y 476.127,Z 314.278,A -85,B 0,C 180,E1 -7411.756,E2 -7411.756} C_VEL
LIN {X 0,Y 476.25,Z 302.274,A -85,B 0,C 180,E1 -7412.058,E2 -7412.058} C_VEL
LIN {X 0,Y 476.856,Z 237.295,A -85,B 0,C 180,E1 -7413.133,E2 -7413.133} C_VEL
LIN {X 0,Y 475.004,Z 226.404,A -85,B 0,C 180,E1 -7413.393,E2 -7413.393} C_VEL
LIN {X 0,Y 474.984,Z 220.607,A -85,B 0,C 180,E1 -7414.468,E2 -7414.468} C_VEL
LIN {X 0,Y 475.309,Z 206.129,A -85,B 0,C 180,E1 -7417.317,E2 -7417.317} C_VEL
LIN {X 0,Y 475.503,Z 190.96,A -85,B 0,C 180,E1 -7420.343,E2 -7420.343} C_VEL
LIN {X 0,Y 474.702,Z 185.55,A -85,B 0,C 180,E1 -7421.494,E2 -7421.494} C_VEL
LIN {X 0,Y 474.624,Z 185.363,A -85,B 0,C 180,E1 -7422.377,E2 -7422.377} C_VEL
LIN {X 0,Y 473.927,Z 185.449,A -85,B 0,C 180,E1 -7423.085,E2 -7423.085} C_VEL
